REGION Network 2: CURRENT MODEL NAME SHOWN IN HMI
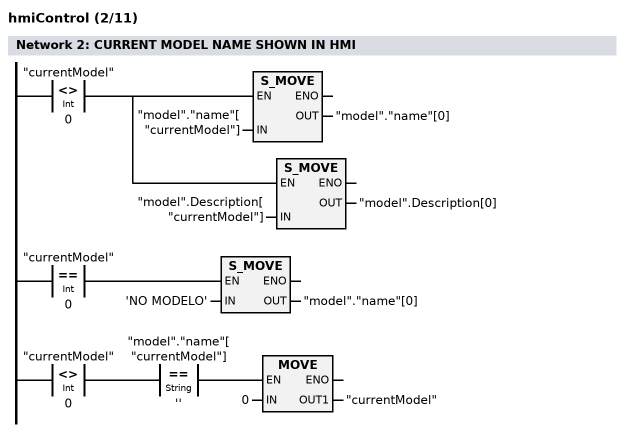
   RUNG wire#powerrail
      { S7_Templates := "SrcType := Int" } NE_Contact(in1 := "currentModel", in2 := 0)
      wire#w1
      S_Move(in := "model"."name"["currentModel"], out => "model"."name"[0])
   END_RUNG
   RUNG wire#w1
      S_Move(in := "model".Description["currentModel"], out => "model".Description[0])
   END_RUNG
   RUNG wire#powerrail
      { S7_Templates := "SrcType := Int" } EQ_Contact(in1 := "currentModel", in2 := 0)
      S_Move(in := 'NO MODELO', out => "model"."name"[0])
   END_RUNG
   RUNG wire#powerrail
      { S7_Templates := "SrcType := Int" } NE_Contact(in1 := "currentModel", in2 := 0)
      { S7_Templates := "SrcType := String" } EQ_Contact(in1 := "model"."name"["currentModel"], in2 := '')
      Move(in := 0, out1 => "currentModel")
   END_RUNG
   // the same network as SCL:
   IF "currentModel" <> 0 THEN
       "model"."name"[0] := "model"."name"["currentModel"];
       "model".Description[0] := "model".Description["currentModel"];
   END_IF;
   IF "currentModel" = 0 THEN "model"."name"[0] := 'NO MODELO'; END_IF;
   IF ("currentModel" <> 0) AND ("model"."name"["currentModel"] = '') THEN "currentModel" := 0; END_IF;
END_REGION

REGION Network 3: MODEL CHANGE (VARIABLE ACTUALIZATION)
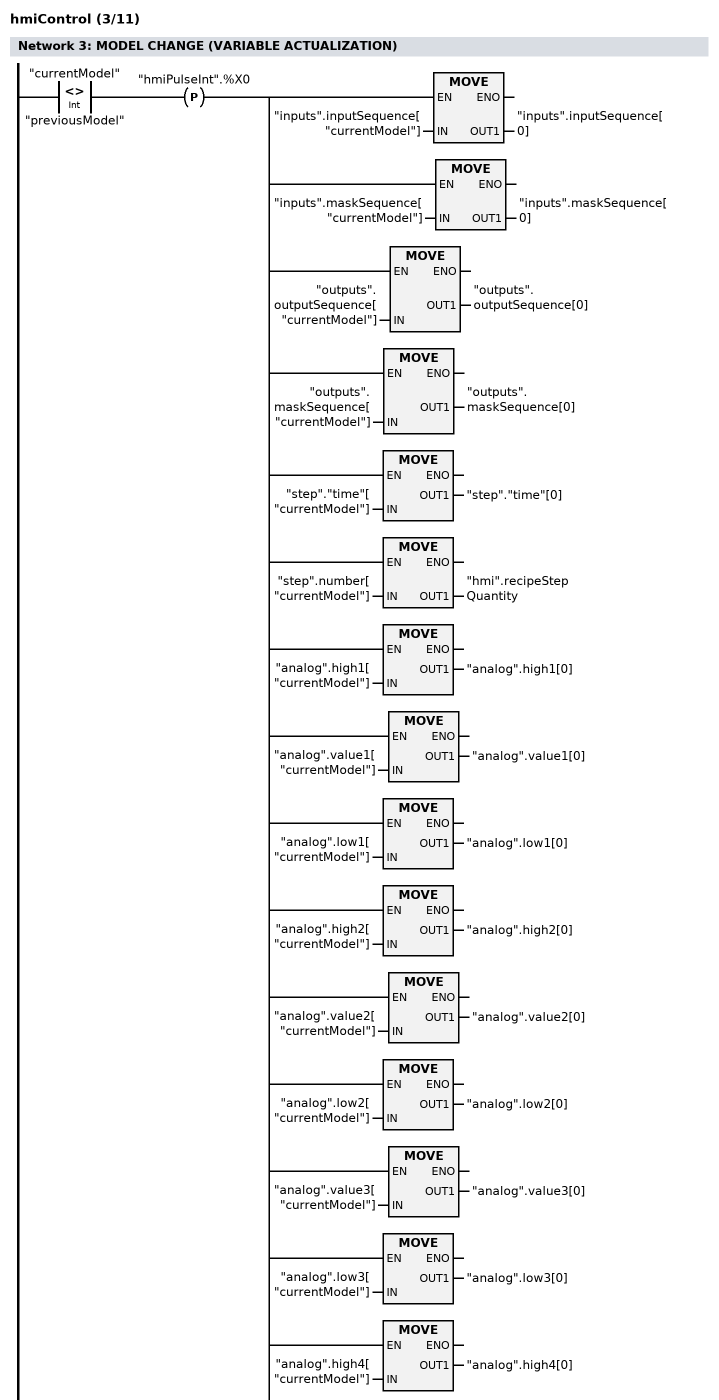
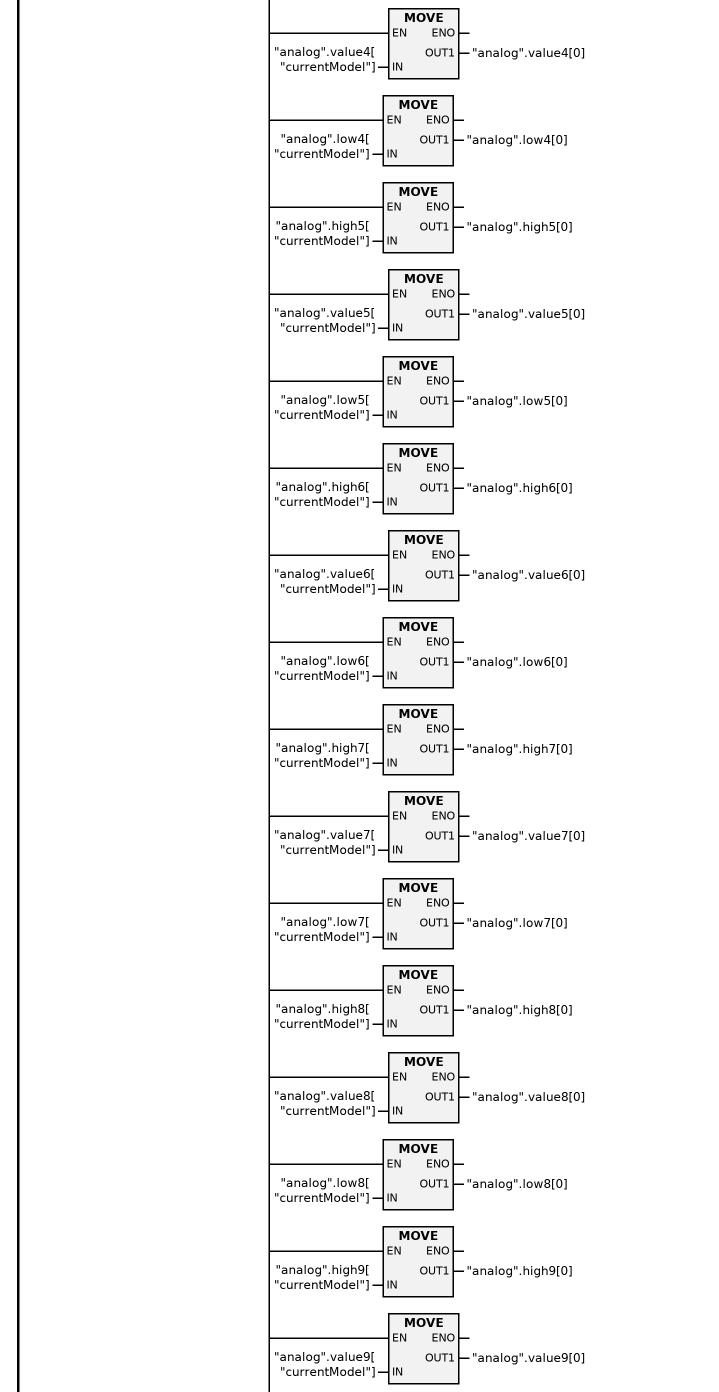
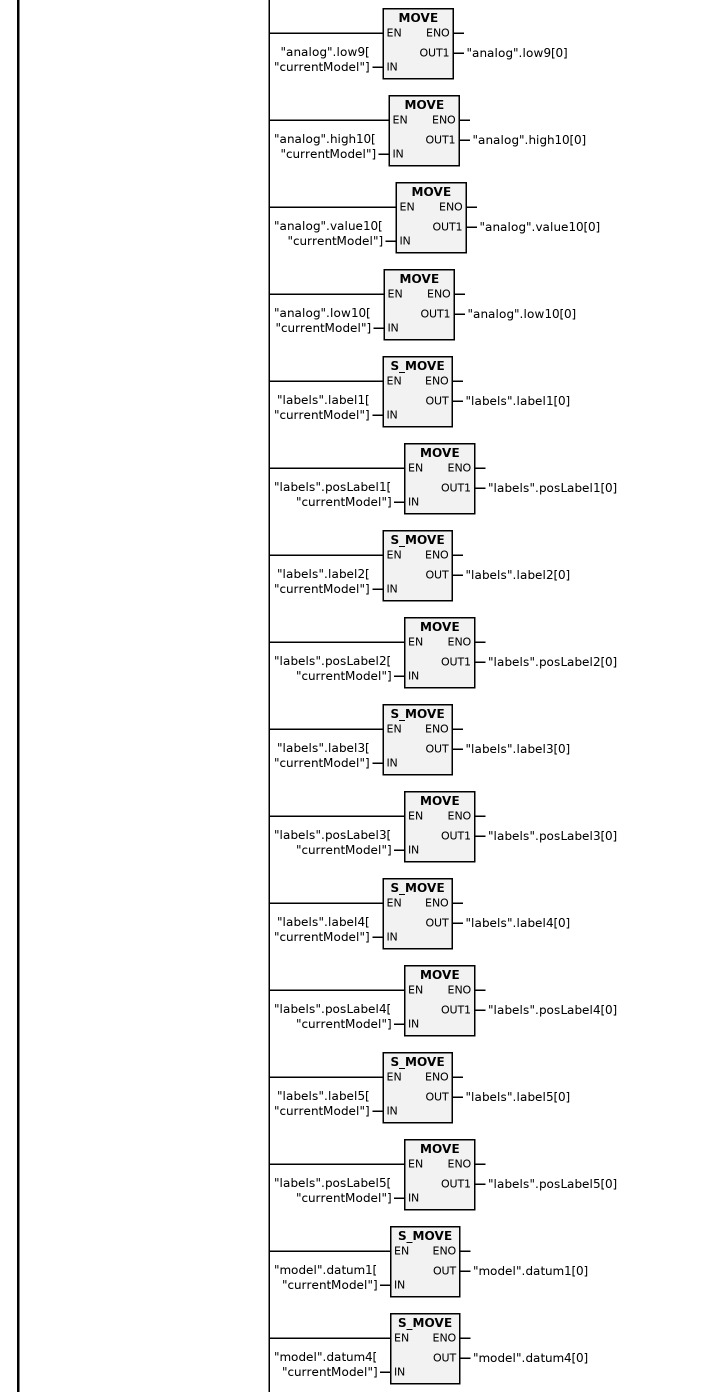
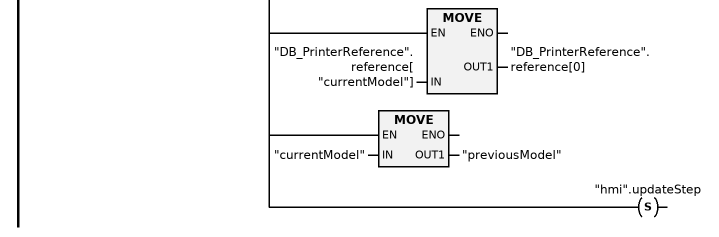
   RUNG wire#powerrail
      { S7_Templates := "SrcType := Int" } NE_Contact(in1 := "currentModel", in2 := "previousModel")
      P_Trig( "hmiPulseInt".%X0 )
      wire#w1
      Move(in := "inputs".inputSequence["currentModel"], out1 => "inputs".inputSequence[0])
   END_RUNG
   RUNG wire#w1
      Move(in := "inputs".maskSequence["currentModel"], out1 => "inputs".maskSequence[0])
   END_RUNG
   RUNG wire#w1
      Move(in := "outputs".outputSequence["currentModel"], out1 => "outputs".outputSequence[0])
   END_RUNG
   RUNG wire#w1
      Move(in := "outputs".maskSequence["currentModel"], out1 => "outputs".maskSequence[0])
   END_RUNG
   RUNG wire#w1
      Move(in := "step"."time"["currentModel"], out1 => "step"."time"[0])
   END_RUNG
   RUNG wire#w1
      Move(in := "step".number["currentModel"], out1 => "hmi".recipeStepQuantity)
   END_RUNG
   RUNG wire#w1
      Move(in := "analog".high1["currentModel"], out1 => "analog".high1[0])
   END_RUNG
   RUNG wire#w1
      Move(in := "analog".value1["currentModel"], out1 => "analog".value1[0])
   END_RUNG
   RUNG wire#w1
      Move(in := "analog".low1["currentModel"], out1 => "analog".low1[0])
   END_RUNG
   RUNG wire#w1
      Move(in := "analog".high2["currentModel"], out1 => "analog".high2[0])
   END_RUNG
   RUNG wire#w1
      Move(in := "analog".value2["currentModel"], out1 => "analog".value2[0])
   END_RUNG
   RUNG wire#w1
      Move(in := "analog".low2["currentModel"], out1 => "analog".low2[0])
   END_RUNG
   RUNG wire#w1
      Move(in := "analog".value3["currentModel"], out1 => "analog".value3[0])
   END_RUNG
   RUNG wire#w1
      Move(in := "analog".low3["currentModel"], out1 => "analog".low3[0])
   END_RUNG
   RUNG wire#w1
      Move(in := "analog".high4["currentModel"], out1 => "analog".high4[0])
   END_RUNG
   RUNG wire#w1
      Move(in := "analog".value4["currentModel"], out1 => "analog".value4[0])
   END_RUNG
   RUNG wire#w1
      Move(in := "analog".low4["currentModel"], out1 => "analog".low4[0])
   END_RUNG
   RUNG wire#w1
      Move(in := "analog".high5["currentModel"], out1 => "analog".high5[0])
   END_RUNG
   RUNG wire#w1
      Move(in := "analog".value5["currentModel"], out1 => "analog".value5[0])
   END_RUNG
   RUNG wire#w1
      Move(in := "analog".low5["currentModel"], out1 => "analog".low5[0])
   END_RUNG
   RUNG wire#w1
      Move(in := "analog".high6["currentModel"], out1 => "analog".high6[0])
   END_RUNG
   RUNG wire#w1
      Move(in := "analog".value6["currentModel"], out1 => "analog".value6[0])
   END_RUNG
   RUNG wire#w1
      Move(in := "analog".low6["currentModel"], out1 => "analog".low6[0])
   END_RUNG
   RUNG wire#w1
      Move(in := "analog".high7["currentModel"], out1 => "analog".high7[0])
   END_RUNG
   RUNG wire#w1
      Move(in := "analog".value7["currentModel"], out1 => "analog".value7[0])
   END_RUNG
   RUNG wire#w1
      Move(in := "analog".low7["currentModel"], out1 => "analog".low7[0])
   END_RUNG
   RUNG wire#w1
      Move(in := "analog".high8["currentModel"], out1 => "analog".high8[0])
   END_RUNG
   RUNG wire#w1
      Move(in := "analog".value8["currentModel"], out1 => "analog".value8[0])
   END_RUNG
   RUNG wire#w1
      Move(in := "analog".low8["currentModel"], out1 => "analog".low8[0])
   END_RUNG
   RUNG wire#w1
      Move(in := "analog".high9["currentModel"], out1 => "analog".high9[0])
   END_RUNG
   RUNG wire#w1
      Move(in := "analog".value9["currentModel"], out1 => "analog".value9[0])
   END_RUNG
   RUNG wire#w1
      Move(in := "analog".low9["currentModel"], out1 => "analog".low9[0])
   END_RUNG
   RUNG wire#w1
      Move(in := "analog".high10["currentModel"], out1 => "analog".high10[0])
   END_RUNG
   RUNG wire#w1
      Move(in := "analog".value10["currentModel"], out1 => "analog".value10[0])
   END_RUNG
   RUNG wire#w1
      Move(in := "analog".low10["currentModel"], out1 => "analog".low10[0])
   END_RUNG
   RUNG wire#w1
      S_Move(in := "labels".label1["currentModel"], out => "labels".label1[0])
   END_RUNG
   RUNG wire#w1
      Move(in := "labels".posLabel1["currentModel"], out1 => "labels".posLabel1[0])
   END_RUNG
   RUNG wire#w1
      S_Move(in := "labels".label2["currentModel"], out => "labels".label2[0])
   END_RUNG
   RUNG wire#w1
      Move(in := "labels".posLabel2["currentModel"], out1 => "labels".posLabel2[0])
   END_RUNG
   RUNG wire#w1
      S_Move(in := "labels".label3["currentModel"], out => "labels".label3[0])
   END_RUNG
   RUNG wire#w1
      Move(in := "labels".posLabel3["currentModel"], out1 => "labels".posLabel3[0])
   END_RUNG
   RUNG wire#w1
      S_Move(in := "labels".label4["currentModel"], out => "labels".label4[0])
   END_RUNG
   RUNG wire#w1
      Move(in := "labels".posLabel4["currentModel"], out1 => "labels".posLabel4[0])
   END_RUNG
   RUNG wire#w1
      S_Move(in := "labels".label5["currentModel"], out => "labels".label5[0])
   END_RUNG
   RUNG wire#w1
      Move(in := "labels".posLabel5["currentModel"], out1 => "labels".posLabel5[0])
   END_RUNG
   RUNG wire#w1
      S_Move(in := "model".datum1["currentModel"], out => "model".datum1[0])
   END_RUNG
   RUNG wire#w1
      S_Move(in := "model".datum4["currentModel"], out => "model".datum4[0])
   END_RUNG
   RUNG wire#w1
      Move(in := "DB_PrinterReference".reference["currentModel"], out1 => "DB_PrinterReference".reference[0])
   END_RUNG
   RUNG wire#w1
      Move(in := "currentModel", out1 => "previousModel")
   END_RUNG
   RUNG wire#w1
      S_Coil( "hmi".updateStep )
   END_RUNG
   // the same network as SCL:
   #_w1 := "currentModel" <> "previousModel";
   #_w2 := #_w1 AND NOT "hmiPulseInt".%X0;   // rising edge
   "hmiPulseInt".%X0 := #_w1;
   IF #_w2 THEN
       "inputs".inputSequence[0] := "inputs".inputSequence["currentModel"];
       "inputs".maskSequence[0] := "inputs".maskSequence["currentModel"];
       "outputs".outputSequence[0] := "outputs".outputSequence["currentModel"];
       "outputs".maskSequence[0] := "outputs".maskSequence["currentModel"];
       "step"."time"[0] := "step"."time"["currentModel"];
       "hmi".recipeStepQuantity := "step".number["currentModel"];
       "analog".high1[0] := "analog".high1["currentModel"];
       "analog".value1[0] := "analog".value1["currentModel"];
       "analog".low1[0] := "analog".low1["currentModel"];
       "analog".high2[0] := "analog".high2["currentModel"];
       "analog".value2[0] := "analog".value2["currentModel"];
       "analog".low2[0] := "analog".low2["currentModel"];
       "analog".value3[0] := "analog".value3["currentModel"];
       "analog".low3[0] := "analog".low3["currentModel"];
       "analog".high4[0] := "analog".high4["currentModel"];
       "analog".value4[0] := "analog".value4["currentModel"];
       "analog".low4[0] := "analog".low4["currentModel"];
       "analog".high5[0] := "analog".high5["currentModel"];
       "analog".value5[0] := "analog".value5["currentModel"];
       "analog".low5[0] := "analog".low5["currentModel"];
       "analog".high6[0] := "analog".high6["currentModel"];
       "analog".value6[0] := "analog".value6["currentModel"];
       "analog".low6[0] := "analog".low6["currentModel"];
       "analog".high7[0] := "analog".high7["currentModel"];
       "analog".value7[0] := "analog".value7["currentModel"];
       "analog".low7[0] := "analog".low7["currentModel"];
       "analog".high8[0] := "analog".high8["currentModel"];
       "analog".value8[0] := "analog".value8["currentModel"];
       "analog".low8[0] := "analog".low8["currentModel"];
       "analog".high9[0] := "analog".high9["currentModel"];
       "analog".value9[0] := "analog".value9["currentModel"];
       "analog".low9[0] := "analog".low9["currentModel"];
       "analog".high10[0] := "analog".high10["currentModel"];
       "analog".value10[0] := "analog".value10["currentModel"];
       "analog".low10[0] := "analog".low10["currentModel"];
       "labels".label1[0] := "labels".label1["currentModel"];
       "labels".posLabel1[0] := "labels".posLabel1["currentModel"];
       "labels".label2[0] := "labels".label2["currentModel"];
       "labels".posLabel2[0] := "labels".posLabel2["currentModel"];
       "labels".label3[0] := "labels".label3["currentModel"];
       "labels".posLabel3[0] := "labels".posLabel3["currentModel"];
       "labels".label4[0] := "labels".label4["currentModel"];
       "labels".posLabel4[0] := "labels".posLabel4["currentModel"];
       "labels".label5[0] := "labels".label5["currentModel"];
       "labels".posLabel5[0] := "labels".posLabel5["currentModel"];
       "model".datum1[0] := "model".datum1["currentModel"];
       "model".datum4[0] := "model".datum4["currentModel"];
       "DB_PrinterReference".reference[0] := "DB_PrinterReference".reference["currentModel"];
       "previousModel" := "currentModel";
       "hmi".updateStep := TRUE;
   END_IF;
END_REGION

REGION Network 4: STEP CHANGE IN RECIPE
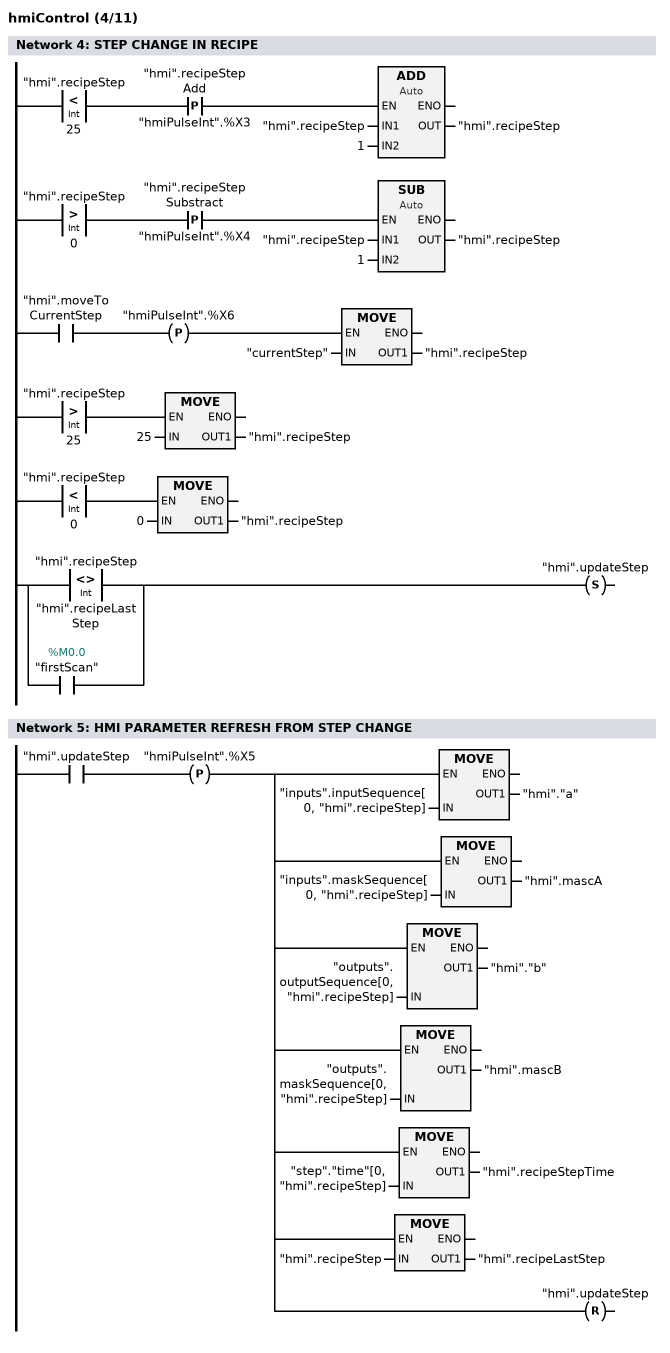
   RUNG wire#powerrail
      { S7_Templates := "SrcType := Int" } LT_Contact(in1 := "hmi".recipeStep, in2 := 25)
      P_Contact(operand := "hmi".recipeStepAdd, bit := "hmiPulseInt".%X3)
      Add(in1 := "hmi".recipeStep, in2 := 1, out => "hmi".recipeStep)
   END_RUNG
   RUNG wire#powerrail
      { S7_Templates := "SrcType := Int" } GT_Contact(in1 := "hmi".recipeStep, in2 := 0)
      P_Contact(operand := "hmi".recipeStepSubstract, bit := "hmiPulseInt".%X4)
      Sub(in1 := "hmi".recipeStep, in2 := 1, out => "hmi".recipeStep)
   END_RUNG
   RUNG wire#powerrail
      Contact( "hmi".moveToCurrentStep )
      P_Trig( "hmiPulseInt".%X6 )
      Move(in := "currentStep", out1 => "hmi".recipeStep)
   END_RUNG
   RUNG wire#powerrail
      { S7_Templates := "SrcType := Int" } GT_Contact(in1 := "hmi".recipeStep, in2 := 25)
      Move(in := 25, out1 => "hmi".recipeStep)
   END_RUNG
   RUNG wire#powerrail
      { S7_Templates := "SrcType := Int" } LT_Contact(in1 := "hmi".recipeStep, in2 := 0)
      Move(in := 0, out1 => "hmi".recipeStep)
   END_RUNG
   RUNG wire#powerrail
      { S7_Templates := "SrcType := Int" } NE_Contact(in1 := "hmi".recipeStep, in2 := "hmi".recipeLastStep)
      wire#w1
      S_Coil( "hmi".updateStep )
   END_RUNG
   RUNG wire#powerrail
      Contact( "firstScan" )
   END_RUNG wire#w1
   // the same network as SCL:
   #_w1 := ("hmi".recipeStep < 25) AND "hmi".recipeStepAdd AND NOT "hmiPulseInt".%X3;   // rising edge of "hmi".recipeStepAdd
   "hmiPulseInt".%X3 := "hmi".recipeStepAdd;
   IF #_w1 THEN "hmi".recipeStep := "hmi".recipeStep + 1; END_IF;
   #_w2 := ("hmi".recipeStep > 0) AND "hmi".recipeStepSubstract AND NOT "hmiPulseInt".%X4;   // rising edge of "hmi".recipeStepSubstract
   "hmiPulseInt".%X4 := "hmi".recipeStepSubstract;
   IF #_w2 THEN "hmi".recipeStep := "hmi".recipeStep - 1; END_IF;
   #_w3 := "hmi".moveToCurrentStep AND NOT "hmiPulseInt".%X6;   // rising edge
   "hmiPulseInt".%X6 := "hmi".moveToCurrentStep;
   IF #_w3 THEN "hmi".recipeStep := "currentStep"; END_IF;
   IF "hmi".recipeStep > 25 THEN "hmi".recipeStep := 25; END_IF;
   IF "hmi".recipeStep < 0 THEN "hmi".recipeStep := 0; END_IF;
   IF ("hmi".recipeStep <> "hmi".recipeLastStep) OR "firstScan" THEN "hmi".updateStep := TRUE; END_IF;
END_REGION

REGION Network 5: HMI PARAMETER REFRESH FROM STEP CHANGE
   RUNG wire#powerrail
      Contact( "hmi".updateStep )
      P_Trig( "hmiPulseInt".%X5 )
      wire#w1
      Move(in := "inputs".inputSequence[0, "hmi".recipeStep], out1 => "hmi"."a")
   END_RUNG
   RUNG wire#w1
      Move(in := "inputs".maskSequence[0, "hmi".recipeStep], out1 => "hmi".mascA)
   END_RUNG
   RUNG wire#w1
      Move(in := "outputs".outputSequence[0, "hmi".recipeStep], out1 => "hmi"."b")
   END_RUNG
   RUNG wire#w1
      Move(in := "outputs".maskSequence[0, "hmi".recipeStep], out1 => "hmi".mascB)
   END_RUNG
   RUNG wire#w1
      Move(in := "step"."time"[0, "hmi".recipeStep], out1 => "hmi".recipeStepTime)
   END_RUNG
   RUNG wire#w1
      Move(in := "hmi".recipeStep, out1 => "hmi".recipeLastStep)
   END_RUNG
   RUNG wire#w1
      R_Coil( "hmi".updateStep )
   END_RUNG
   // the same network as SCL:
   #_w1 := "hmi".updateStep AND NOT "hmiPulseInt".%X5;   // rising edge
   "hmiPulseInt".%X5 := "hmi".updateStep;
   IF #_w1 THEN
       "hmi"."a" := "inputs".inputSequence[0, "hmi".recipeStep];
       "hmi".mascA := "inputs".maskSequence[0, "hmi".recipeStep];
       "hmi"."b" := "outputs".outputSequence[0, "hmi".recipeStep];
       "hmi".mascB := "outputs".maskSequence[0, "hmi".recipeStep];
       "hmi".recipeStepTime := "step"."time"[0, "hmi".recipeStep];
       "hmi".recipeLastStep := "hmi".recipeStep;
       "hmi".updateStep := FALSE;
   END_IF;
END_REGION

REGION Network 6: EDIT VALUES IN CURRENT RECIPE
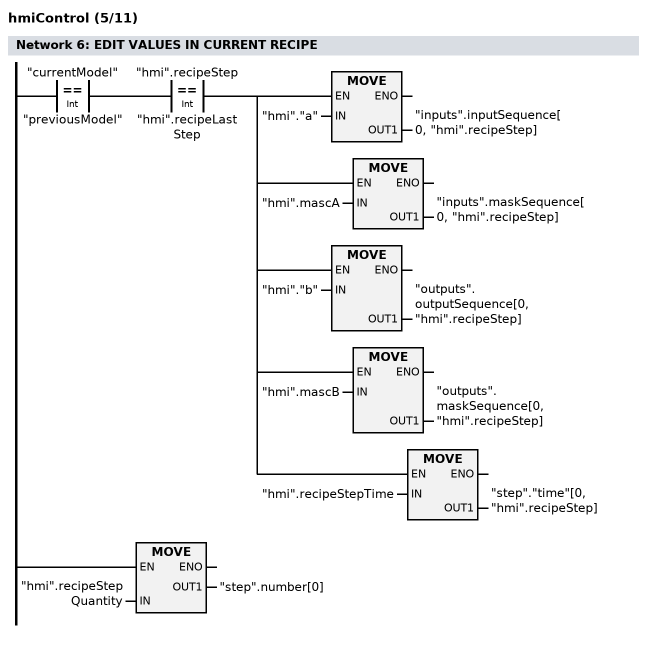
   RUNG wire#powerrail
      { S7_Templates := "SrcType := Int" } EQ_Contact(in1 := "currentModel", in2 := "previousModel")
      { S7_Templates := "SrcType := Int" } EQ_Contact(in1 := "hmi".recipeStep, in2 := "hmi".recipeLastStep)
      wire#w1
      Move(in := "hmi"."a", out1 => "inputs".inputSequence[0, "hmi".recipeStep])
   END_RUNG
   RUNG wire#w1
      Move(in := "hmi".mascA, out1 => "inputs".maskSequence[0, "hmi".recipeStep])
   END_RUNG
   RUNG wire#w1
      Move(in := "hmi"."b", out1 => "outputs".outputSequence[0, "hmi".recipeStep])
   END_RUNG
   RUNG wire#w1
      Move(in := "hmi".mascB, out1 => "outputs".maskSequence[0, "hmi".recipeStep])
   END_RUNG
   RUNG wire#w1
      Move(in := "hmi".recipeStepTime, out1 => "step"."time"[0, "hmi".recipeStep])
   END_RUNG
   RUNG wire#powerrail
      Move(in := "hmi".recipeStepQuantity, out1 => "step".number[0])
   END_RUNG
   // the same network as SCL:
   #_w1 := ("currentModel" = "previousModel") AND ("hmi".recipeStep = "hmi".recipeLastStep);
   IF #_w1 THEN
       "inputs".inputSequence[0, "hmi".recipeStep] := "hmi"."a";
       "inputs".maskSequence[0, "hmi".recipeStep] := "hmi".mascA;
       "outputs".outputSequence[0, "hmi".recipeStep] := "hmi"."b";
       "outputs".maskSequence[0, "hmi".recipeStep] := "hmi".mascB;
       "step"."time"[0, "hmi".recipeStep] := "hmi".recipeStepTime;
   END_IF;
   "step".number[0] := "hmi".recipeStepQuantity;
END_REGION

REGION Network 7: WRITE AND READ IN SCREEN
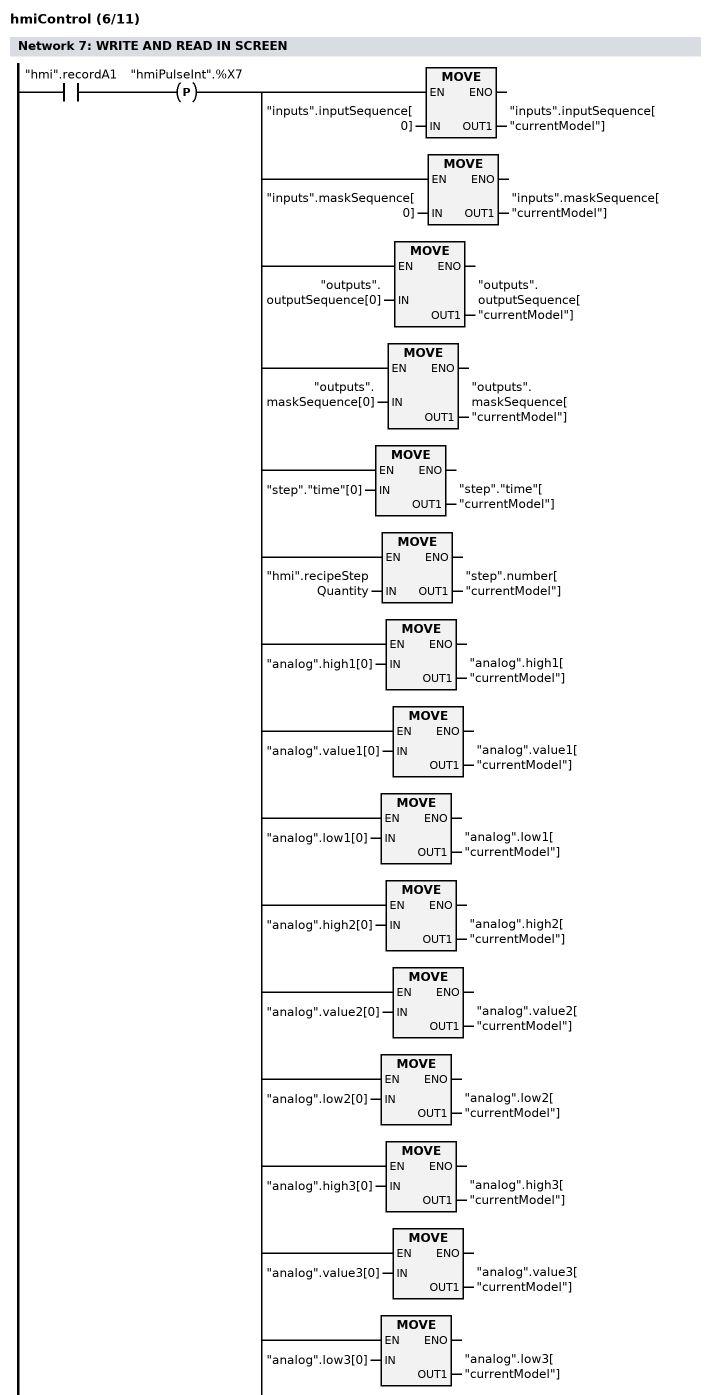
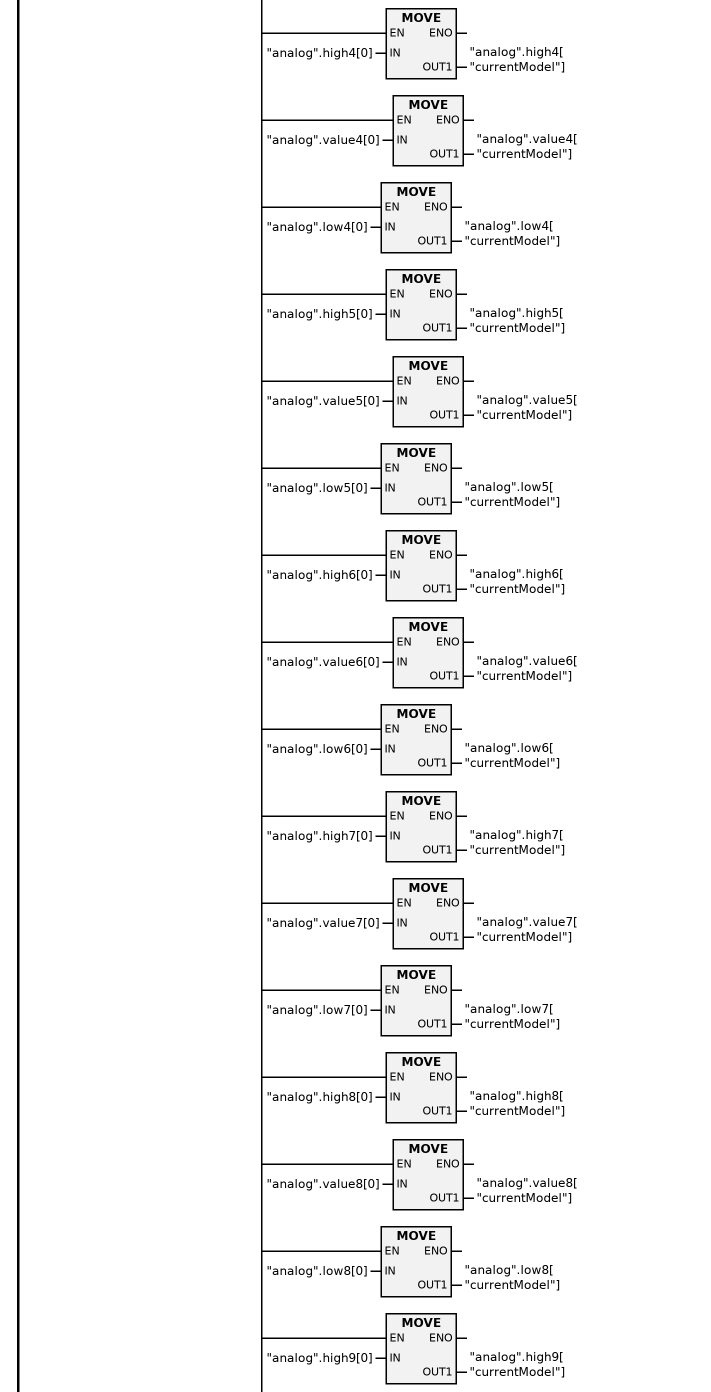
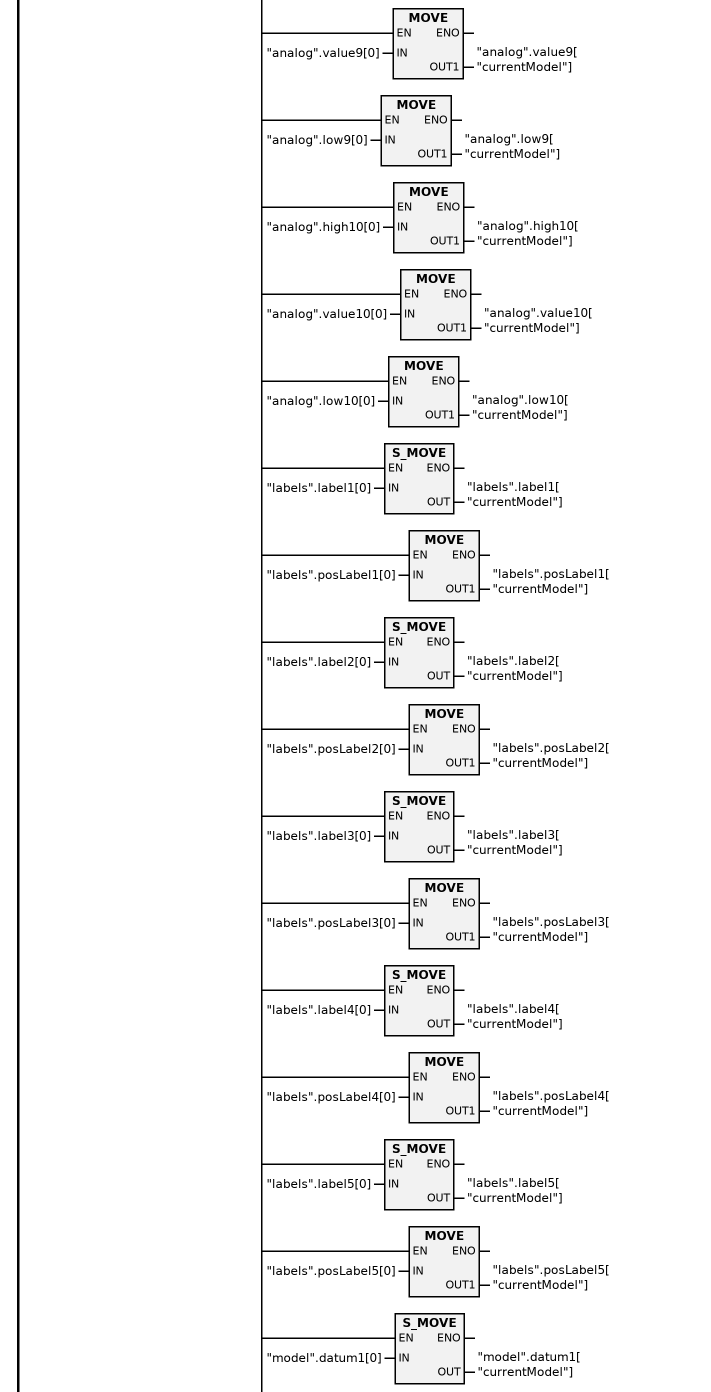
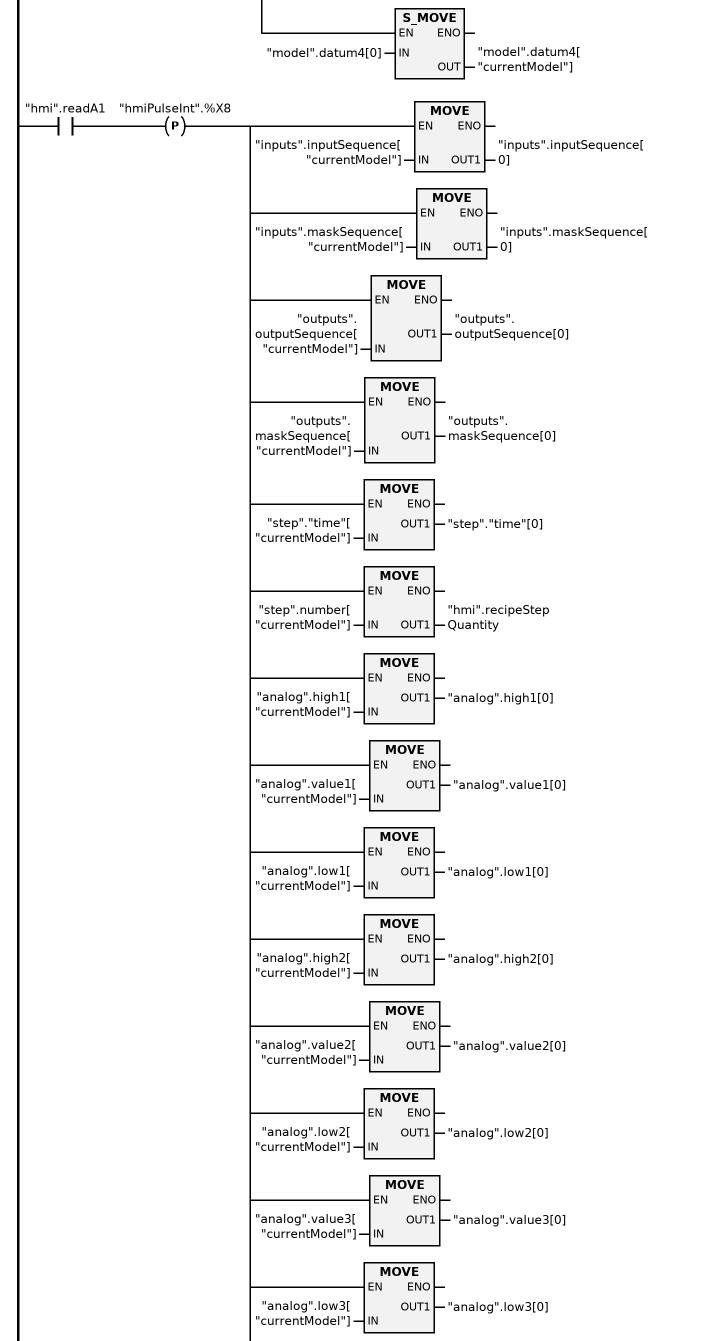
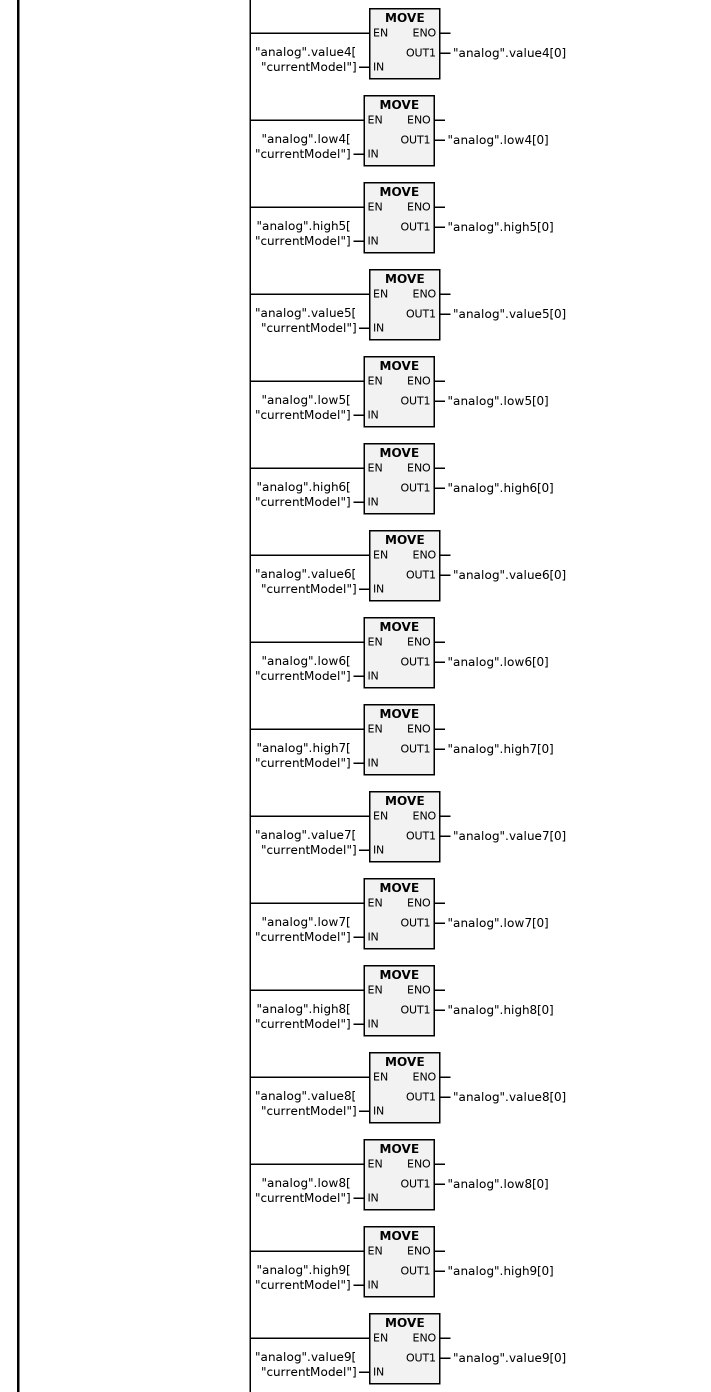
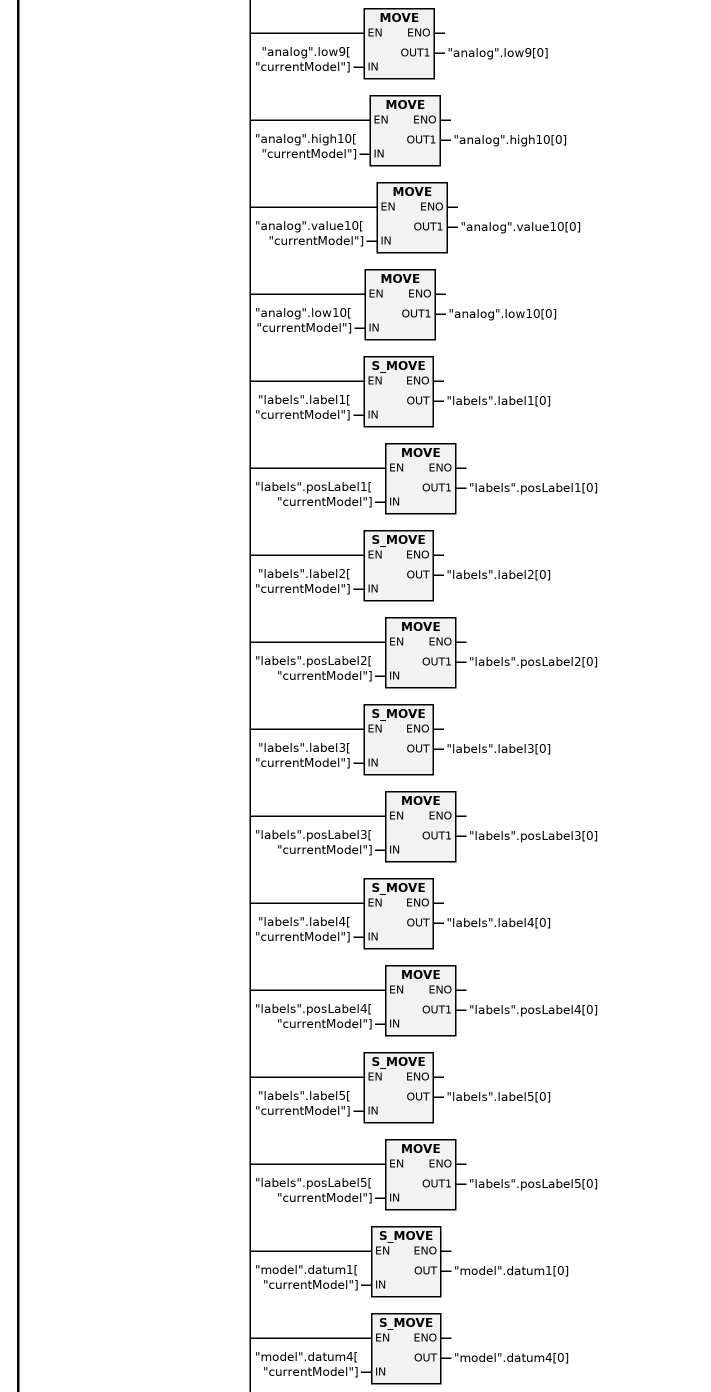
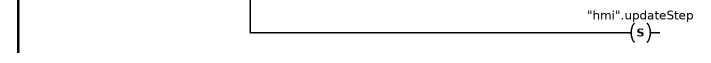
   RUNG wire#powerrail
      Contact( "hmi".recordA1 )
      P_Trig( "hmiPulseInt".%X7 )
      wire#w1
      Move(in := "inputs".inputSequence[0], out1 => "inputs".inputSequence["currentModel"])
   END_RUNG
   RUNG wire#w1
      Move(in := "inputs".maskSequence[0], out1 => "inputs".maskSequence["currentModel"])
   END_RUNG
   RUNG wire#w1
      Move(in := "outputs".outputSequence[0], out1 => "outputs".outputSequence["currentModel"])
   END_RUNG
   RUNG wire#w1
      Move(in := "outputs".maskSequence[0], out1 => "outputs".maskSequence["currentModel"])
   END_RUNG
   RUNG wire#w1
      Move(in := "step"."time"[0], out1 => "step"."time"["currentModel"])
   END_RUNG
   RUNG wire#w1
      Move(in := "hmi".recipeStepQuantity, out1 => "step".number["currentModel"])
   END_RUNG
   RUNG wire#w1
      Move(in := "analog".high1[0], out1 => "analog".high1["currentModel"])
   END_RUNG
   RUNG wire#w1
      Move(in := "analog".value1[0], out1 => "analog".value1["currentModel"])
   END_RUNG
   RUNG wire#w1
      Move(in := "analog".low1[0], out1 => "analog".low1["currentModel"])
   END_RUNG
   RUNG wire#w1
      Move(in := "analog".high2[0], out1 => "analog".high2["currentModel"])
   END_RUNG
   RUNG wire#w1
      Move(in := "analog".value2[0], out1 => "analog".value2["currentModel"])
   END_RUNG
   RUNG wire#w1
      Move(in := "analog".low2[0], out1 => "analog".low2["currentModel"])
   END_RUNG
   RUNG wire#w1
      Move(in := "analog".high3[0], out1 => "analog".high3["currentModel"])
   END_RUNG
   RUNG wire#w1
      Move(in := "analog".value3[0], out1 => "analog".value3["currentModel"])
   END_RUNG
   RUNG wire#w1
      Move(in := "analog".low3[0], out1 => "analog".low3["currentModel"])
   END_RUNG
   RUNG wire#w1
      Move(in := "analog".high4[0], out1 => "analog".high4["currentModel"])
   END_RUNG
   RUNG wire#w1
      Move(in := "analog".value4[0], out1 => "analog".value4["currentModel"])
   END_RUNG
   RUNG wire#w1
      Move(in := "analog".low4[0], out1 => "analog".low4["currentModel"])
   END_RUNG
   RUNG wire#w1
      Move(in := "analog".high5[0], out1 => "analog".high5["currentModel"])
   END_RUNG
   RUNG wire#w1
      Move(in := "analog".value5[0], out1 => "analog".value5["currentModel"])
   END_RUNG
   RUNG wire#w1
      Move(in := "analog".low5[0], out1 => "analog".low5["currentModel"])
   END_RUNG
   RUNG wire#w1
      Move(in := "analog".high6[0], out1 => "analog".high6["currentModel"])
   END_RUNG
   RUNG wire#w1
      Move(in := "analog".value6[0], out1 => "analog".value6["currentModel"])
   END_RUNG
   RUNG wire#w1
      Move(in := "analog".low6[0], out1 => "analog".low6["currentModel"])
   END_RUNG
   RUNG wire#w1
      Move(in := "analog".high7[0], out1 => "analog".high7["currentModel"])
   END_RUNG
   RUNG wire#w1
      Move(in := "analog".value7[0], out1 => "analog".value7["currentModel"])
   END_RUNG
   RUNG wire#w1
      Move(in := "analog".low7[0], out1 => "analog".low7["currentModel"])
   END_RUNG
   RUNG wire#w1
      Move(in := "analog".high8[0], out1 => "analog".high8["currentModel"])
   END_RUNG
   RUNG wire#w1
      Move(in := "analog".value8[0], out1 => "analog".value8["currentModel"])
   END_RUNG
   RUNG wire#w1
      Move(in := "analog".low8[0], out1 => "analog".low8["currentModel"])
   END_RUNG
   RUNG wire#w1
      Move(in := "analog".high9[0], out1 => "analog".high9["currentModel"])
   END_RUNG
   RUNG wire#w1
      Move(in := "analog".value9[0], out1 => "analog".value9["currentModel"])
   END_RUNG
   RUNG wire#w1
      Move(in := "analog".low9[0], out1 => "analog".low9["currentModel"])
   END_RUNG
   RUNG wire#w1
      Move(in := "analog".high10[0], out1 => "analog".high10["currentModel"])
   END_RUNG
   RUNG wire#w1
      Move(in := "analog".value10[0], out1 => "analog".value10["currentModel"])
   END_RUNG
   RUNG wire#w1
      Move(in := "analog".low10[0], out1 => "analog".low10["currentModel"])
   END_RUNG
   RUNG wire#w1
      S_Move(in := "labels".label1[0], out => "labels".label1["currentModel"])
   END_RUNG
   RUNG wire#w1
      Move(in := "labels".posLabel1[0], out1 => "labels".posLabel1["currentModel"])
   END_RUNG
   RUNG wire#w1
      S_Move(in := "labels".label2[0], out => "labels".label2["currentModel"])
   END_RUNG
   RUNG wire#w1
      Move(in := "labels".posLabel2[0], out1 => "labels".posLabel2["currentModel"])
   END_RUNG
   RUNG wire#w1
      S_Move(in := "labels".label3[0], out => "labels".label3["currentModel"])
   END_RUNG
   RUNG wire#w1
      Move(in := "labels".posLabel3[0], out1 => "labels".posLabel3["currentModel"])
   END_RUNG
   RUNG wire#w1
      S_Move(in := "labels".label4[0], out => "labels".label4["currentModel"])
   END_RUNG
   RUNG wire#w1
      Move(in := "labels".posLabel4[0], out1 => "labels".posLabel4["currentModel"])
   END_RUNG
   RUNG wire#w1
      S_Move(in := "labels".label5[0], out => "labels".label5["currentModel"])
   END_RUNG
   RUNG wire#w1
      Move(in := "labels".posLabel5[0], out1 => "labels".posLabel5["currentModel"])
   END_RUNG
   RUNG wire#w1
      S_Move(in := "model".datum1[0], out => "model".datum1["currentModel"])
   END_RUNG
   RUNG wire#w1
      S_Move(in := "model".datum4[0], out => "model".datum4["currentModel"])
   END_RUNG
   RUNG wire#powerrail
      Contact( "hmi".readA1 )
      P_Trig( "hmiPulseInt".%X8 )
      wire#w2
      Move(in := "inputs".inputSequence["currentModel"], out1 => "inputs".inputSequence[0])
   END_RUNG
   RUNG wire#w2
      Move(in := "inputs".maskSequence["currentModel"], out1 => "inputs".maskSequence[0])
   END_RUNG
   RUNG wire#w2
      Move(in := "outputs".outputSequence["currentModel"], out1 => "outputs".outputSequence[0])
   END_RUNG
   RUNG wire#w2
      Move(in := "outputs".maskSequence["currentModel"], out1 => "outputs".maskSequence[0])
   END_RUNG
   RUNG wire#w2
      Move(in := "step"."time"["currentModel"], out1 => "step"."time"[0])
   END_RUNG
   RUNG wire#w2
      Move(in := "step".number["currentModel"], out1 => "hmi".recipeStepQuantity)
   END_RUNG
   RUNG wire#w2
      Move(in := "analog".high1["currentModel"], out1 => "analog".high1[0])
   END_RUNG
   RUNG wire#w2
      Move(in := "analog".value1["currentModel"], out1 => "analog".value1[0])
   END_RUNG
   RUNG wire#w2
      Move(in := "analog".low1["currentModel"], out1 => "analog".low1[0])
   END_RUNG
   RUNG wire#w2
      Move(in := "analog".high2["currentModel"], out1 => "analog".high2[0])
   END_RUNG
   RUNG wire#w2
      Move(in := "analog".value2["currentModel"], out1 => "analog".value2[0])
   END_RUNG
   RUNG wire#w2
      Move(in := "analog".low2["currentModel"], out1 => "analog".low2[0])
   END_RUNG
   RUNG wire#w2
      Move(in := "analog".value3["currentModel"], out1 => "analog".value3[0])
   END_RUNG
   RUNG wire#w2
      Move(in := "analog".low3["currentModel"], out1 => "analog".low3[0])
   END_RUNG
   RUNG wire#w2
      Move(in := "analog".value4["currentModel"], out1 => "analog".value4[0])
   END_RUNG
   RUNG wire#w2
      Move(in := "analog".low4["currentModel"], out1 => "analog".low4[0])
   END_RUNG
   RUNG wire#w2
      Move(in := "analog".high5["currentModel"], out1 => "analog".high5[0])
   END_RUNG
   RUNG wire#w2
      Move(in := "analog".value5["currentModel"], out1 => "analog".value5[0])
   END_RUNG
   RUNG wire#w2
      Move(in := "analog".low5["currentModel"], out1 => "analog".low5[0])
   END_RUNG
   RUNG wire#w2
      Move(in := "analog".high6["currentModel"], out1 => "analog".high6[0])
   END_RUNG
   RUNG wire#w2
      Move(in := "analog".value6["currentModel"], out1 => "analog".value6[0])
   END_RUNG
   RUNG wire#w2
      Move(in := "analog".low6["currentModel"], out1 => "analog".low6[0])
   END_RUNG
   RUNG wire#w2
      Move(in := "analog".high7["currentModel"], out1 => "analog".high7[0])
   END_RUNG
   RUNG wire#w2
      Move(in := "analog".value7["currentModel"], out1 => "analog".value7[0])
   END_RUNG
   RUNG wire#w2
      Move(in := "analog".low7["currentModel"], out1 => "analog".low7[0])
   END_RUNG
   RUNG wire#w2
      Move(in := "analog".high8["currentModel"], out1 => "analog".high8[0])
   END_RUNG
   RUNG wire#w2
      Move(in := "analog".value8["currentModel"], out1 => "analog".value8[0])
   END_RUNG
   RUNG wire#w2
      Move(in := "analog".low8["currentModel"], out1 => "analog".low8[0])
   END_RUNG
   RUNG wire#w2
      Move(in := "analog".high9["currentModel"], out1 => "analog".high9[0])
   END_RUNG
   RUNG wire#w2
      Move(in := "analog".value9["currentModel"], out1 => "analog".value9[0])
   END_RUNG
   RUNG wire#w2
      Move(in := "analog".low9["currentModel"], out1 => "analog".low9[0])
   END_RUNG
   RUNG wire#w2
      Move(in := "analog".high10["currentModel"], out1 => "analog".high10[0])
   END_RUNG
   RUNG wire#w2
      Move(in := "analog".value10["currentModel"], out1 => "analog".value10[0])
   END_RUNG
   RUNG wire#w2
      Move(in := "analog".low10["currentModel"], out1 => "analog".low10[0])
   END_RUNG
   RUNG wire#w2
      S_Move(in := "labels".label1["currentModel"], out => "labels".label1[0])
   END_RUNG
   RUNG wire#w2
      Move(in := "labels".posLabel1["currentModel"], out1 => "labels".posLabel1[0])
   END_RUNG
   RUNG wire#w2
      S_Move(in := "labels".label2["currentModel"], out => "labels".label2[0])
   END_RUNG
   RUNG wire#w2
      Move(in := "labels".posLabel2["currentModel"], out1 => "labels".posLabel2[0])
   END_RUNG
   RUNG wire#w2
      S_Move(in := "labels".label3["currentModel"], out => "labels".label3[0])
   END_RUNG
   RUNG wire#w2
      Move(in := "labels".posLabel3["currentModel"], out1 => "labels".posLabel3[0])
   END_RUNG
   RUNG wire#w2
      S_Move(in := "labels".label4["currentModel"], out => "labels".label4[0])
   END_RUNG
   RUNG wire#w2
      Move(in := "labels".posLabel4["currentModel"], out1 => "labels".posLabel4[0])
   END_RUNG
   RUNG wire#w2
      S_Move(in := "labels".label5["currentModel"], out => "labels".label5[0])
   END_RUNG
   RUNG wire#w2
      Move(in := "labels".posLabel5["currentModel"], out1 => "labels".posLabel5[0])
   END_RUNG
   RUNG wire#w2
      S_Move(in := "model".datum1["currentModel"], out => "model".datum1[0])
   END_RUNG
   RUNG wire#w2
      S_Move(in := "model".datum4["currentModel"], out => "model".datum4[0])
   END_RUNG
   RUNG wire#w2
      S_Coil( "hmi".updateStep )
   END_RUNG
   // the same network as SCL:
   #_w1 := "hmi".recordA1 AND NOT "hmiPulseInt".%X7;   // rising edge
   "hmiPulseInt".%X7 := "hmi".recordA1;
   IF #_w1 THEN
       "inputs".inputSequence["currentModel"] := "inputs".inputSequence[0];
       "inputs".maskSequence["currentModel"] := "inputs".maskSequence[0];
       "outputs".outputSequence["currentModel"] := "outputs".outputSequence[0];
       "outputs".maskSequence["currentModel"] := "outputs".maskSequence[0];
       "step"."time"["currentModel"] := "step"."time"[0];
       "step".number["currentModel"] := "hmi".recipeStepQuantity;
       "analog".high1["currentModel"] := "analog".high1[0];
       "analog".value1["currentModel"] := "analog".value1[0];
       "analog".low1["currentModel"] := "analog".low1[0];
       "analog".high2["currentModel"] := "analog".high2[0];
       "analog".value2["currentModel"] := "analog".value2[0];
       "analog".low2["currentModel"] := "analog".low2[0];
       "analog".high3["currentModel"] := "analog".high3[0];
       "analog".value3["currentModel"] := "analog".value3[0];
       "analog".low3["currentModel"] := "analog".low3[0];
       "analog".high4["currentModel"] := "analog".high4[0];
       "analog".value4["currentModel"] := "analog".value4[0];
       "analog".low4["currentModel"] := "analog".low4[0];
       "analog".high5["currentModel"] := "analog".high5[0];
       "analog".value5["currentModel"] := "analog".value5[0];
       "analog".low5["currentModel"] := "analog".low5[0];
       "analog".high6["currentModel"] := "analog".high6[0];
       "analog".value6["currentModel"] := "analog".value6[0];
       "analog".low6["currentModel"] := "analog".low6[0];
       "analog".high7["currentModel"] := "analog".high7[0];
       "analog".value7["currentModel"] := "analog".value7[0];
       "analog".low7["currentModel"] := "analog".low7[0];
       "analog".high8["currentModel"] := "analog".high8[0];
       "analog".value8["currentModel"] := "analog".value8[0];
       "analog".low8["currentModel"] := "analog".low8[0];
       "analog".high9["currentModel"] := "analog".high9[0];
       "analog".value9["currentModel"] := "analog".value9[0];
       "analog".low9["currentModel"] := "analog".low9[0];
       "analog".high10["currentModel"] := "analog".high10[0];
       "analog".value10["currentModel"] := "analog".value10[0];
       "analog".low10["currentModel"] := "analog".low10[0];
       "labels".label1["currentModel"] := "labels".label1[0];
       "labels".posLabel1["currentModel"] := "labels".posLabel1[0];
       "labels".label2["currentModel"] := "labels".label2[0];
       "labels".posLabel2["currentModel"] := "labels".posLabel2[0];
       "labels".label3["currentModel"] := "labels".label3[0];
       "labels".posLabel3["currentModel"] := "labels".posLabel3[0];
       "labels".label4["currentModel"] := "labels".label4[0];
       "labels".posLabel4["currentModel"] := "labels".posLabel4[0];
       "labels".label5["currentModel"] := "labels".label5[0];
       "labels".posLabel5["currentModel"] := "labels".posLabel5[0];
       "model".datum1["currentModel"] := "model".datum1[0];
       "model".datum4["currentModel"] := "model".datum4[0];
   END_IF;
   #_w2 := "hmi".readA1 AND NOT "hmiPulseInt".%X8;   // rising edge
   "hmiPulseInt".%X8 := "hmi".readA1;
   IF #_w2 THEN
       "inputs".inputSequence[0] := "inputs".inputSequence["currentModel"];
       "inputs".maskSequence[0] := "inputs".maskSequence["currentModel"];
       "outputs".outputSequence[0] := "outputs".outputSequence["currentModel"];
       "outputs".maskSequence[0] := "outputs".maskSequence["currentModel"];
       "step"."time"[0] := "step"."time"["currentModel"];
       "hmi".recipeStepQuantity := "step".number["currentModel"];
       "analog".high1[0] := "analog".high1["currentModel"];
       "analog".value1[0] := "analog".value1["currentModel"];
       "analog".low1[0] := "analog".low1["currentModel"];
       "analog".high2[0] := "analog".high2["currentModel"];
       "analog".value2[0] := "analog".value2["currentModel"];
       "analog".low2[0] := "analog".low2["currentModel"];
       "analog".value3[0] := "analog".value3["currentModel"];
       "analog".low3[0] := "analog".low3["currentModel"];
       "analog".value4[0] := "analog".value4["currentModel"];
       "analog".low4[0] := "analog".low4["currentModel"];
       "analog".high5[0] := "analog".high5["currentModel"];
       "analog".value5[0] := "analog".value5["currentModel"];
       "analog".low5[0] := "analog".low5["currentModel"];
       "analog".high6[0] := "analog".high6["currentModel"];
       "analog".value6[0] := "analog".value6["currentModel"];
       "analog".low6[0] := "analog".low6["currentModel"];
       "analog".high7[0] := "analog".high7["currentModel"];
       "analog".value7[0] := "analog".value7["currentModel"];
       "analog".low7[0] := "analog".low7["currentModel"];
       "analog".high8[0] := "analog".high8["currentModel"];
       "analog".value8[0] := "analog".value8["currentModel"];
       "analog".low8[0] := "analog".low8["currentModel"];
       "analog".high9[0] := "analog".high9["currentModel"];
       "analog".value9[0] := "analog".value9["currentModel"];
       "analog".low9[0] := "analog".low9["currentModel"];
       "analog".high10[0] := "analog".high10["currentModel"];
       "analog".value10[0] := "analog".value10["currentModel"];
       "analog".low10[0] := "analog".low10["currentModel"];
       "labels".label1[0] := "labels".label1["currentModel"];
       "labels".posLabel1[0] := "labels".posLabel1["currentModel"];
       "labels".label2[0] := "labels".label2["currentModel"];
       "labels".posLabel2[0] := "labels".posLabel2["currentModel"];
       "labels".label3[0] := "labels".label3["currentModel"];
       "labels".posLabel3[0] := "labels".posLabel3["currentModel"];
       "labels".label4[0] := "labels".label4["currentModel"];
       "labels".posLabel4[0] := "labels".posLabel4["currentModel"];
       "labels".label5[0] := "labels".label5["currentModel"];
       "labels".posLabel5[0] := "labels".posLabel5["currentModel"];
       "model".datum1[0] := "model".datum1["currentModel"];
       "model".datum4[0] := "model".datum4["currentModel"];
       "hmi".updateStep := TRUE;
   END_IF;
END_REGION

REGION Network 8: NUMBER OF STEPS OF RECIPE
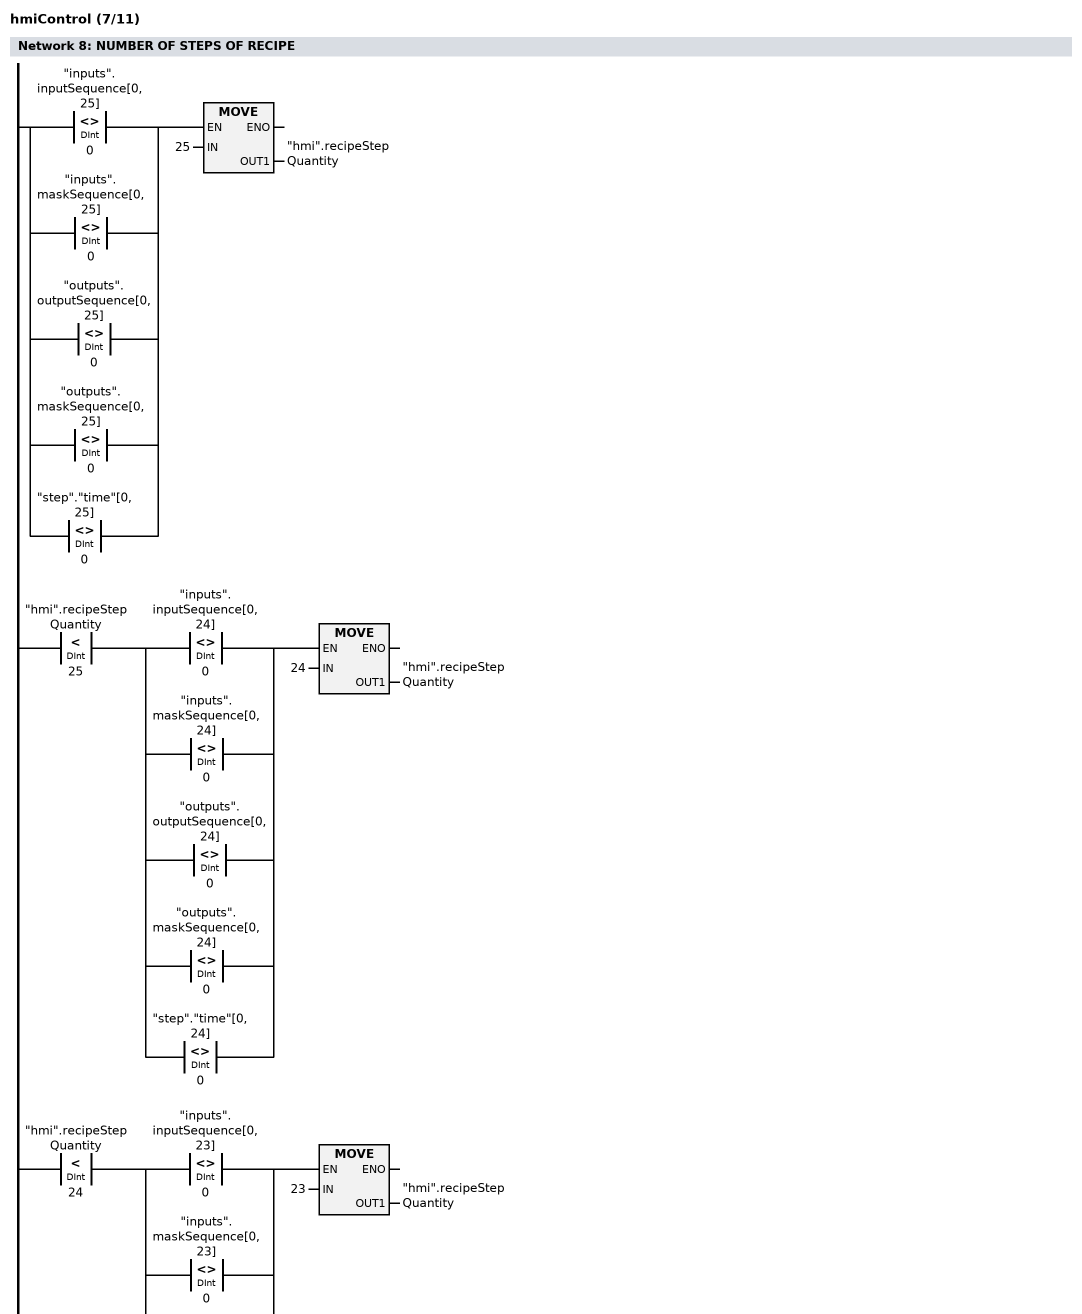
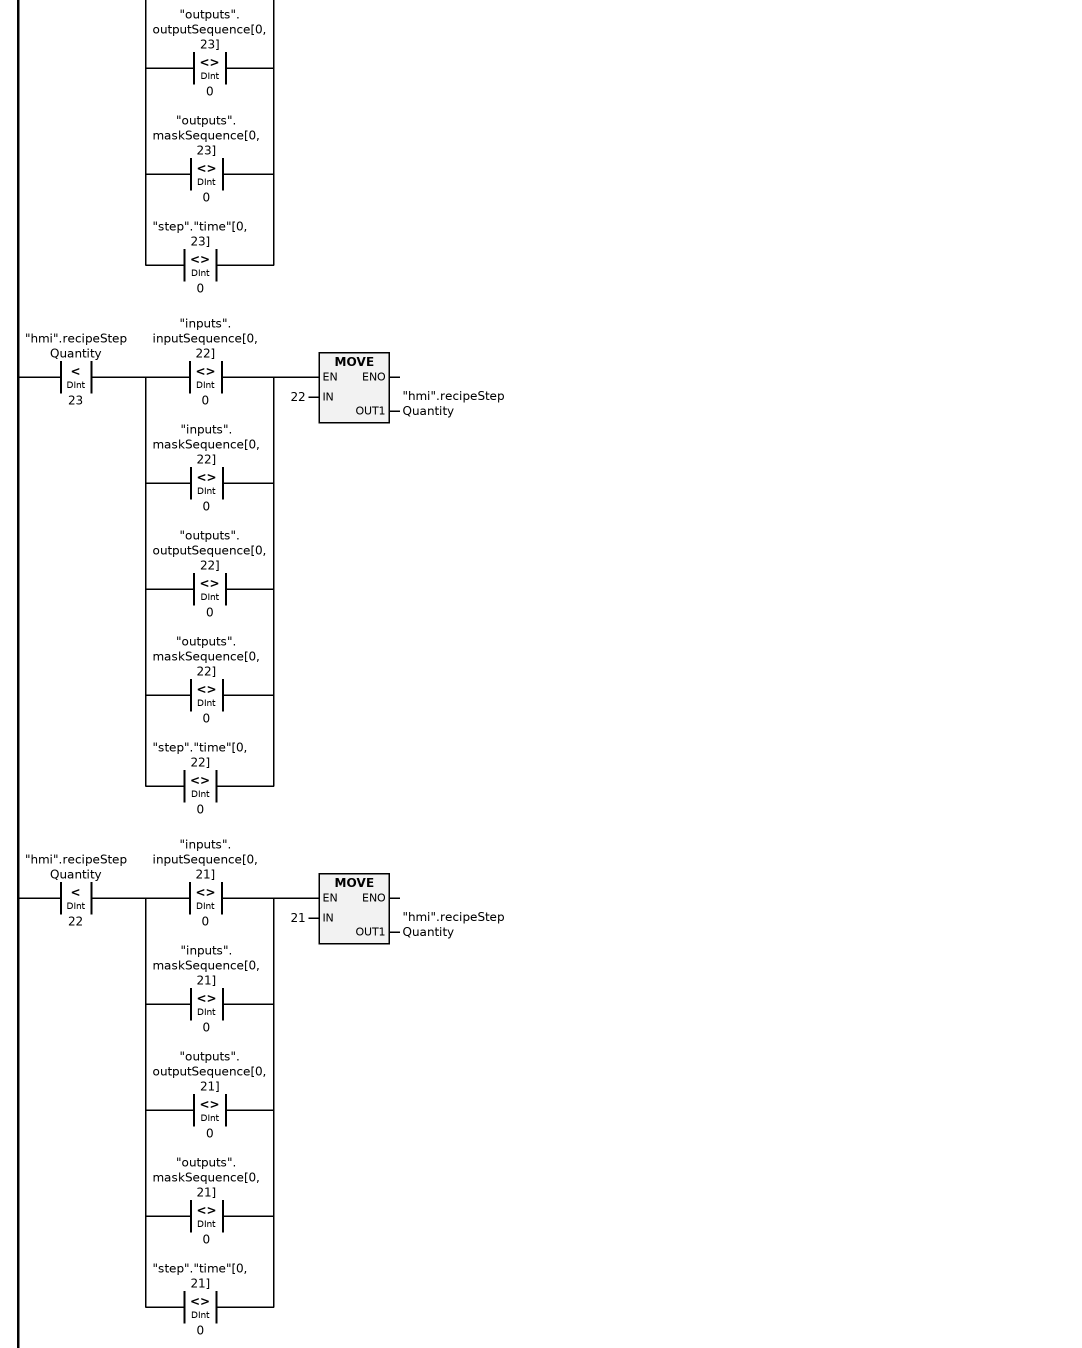
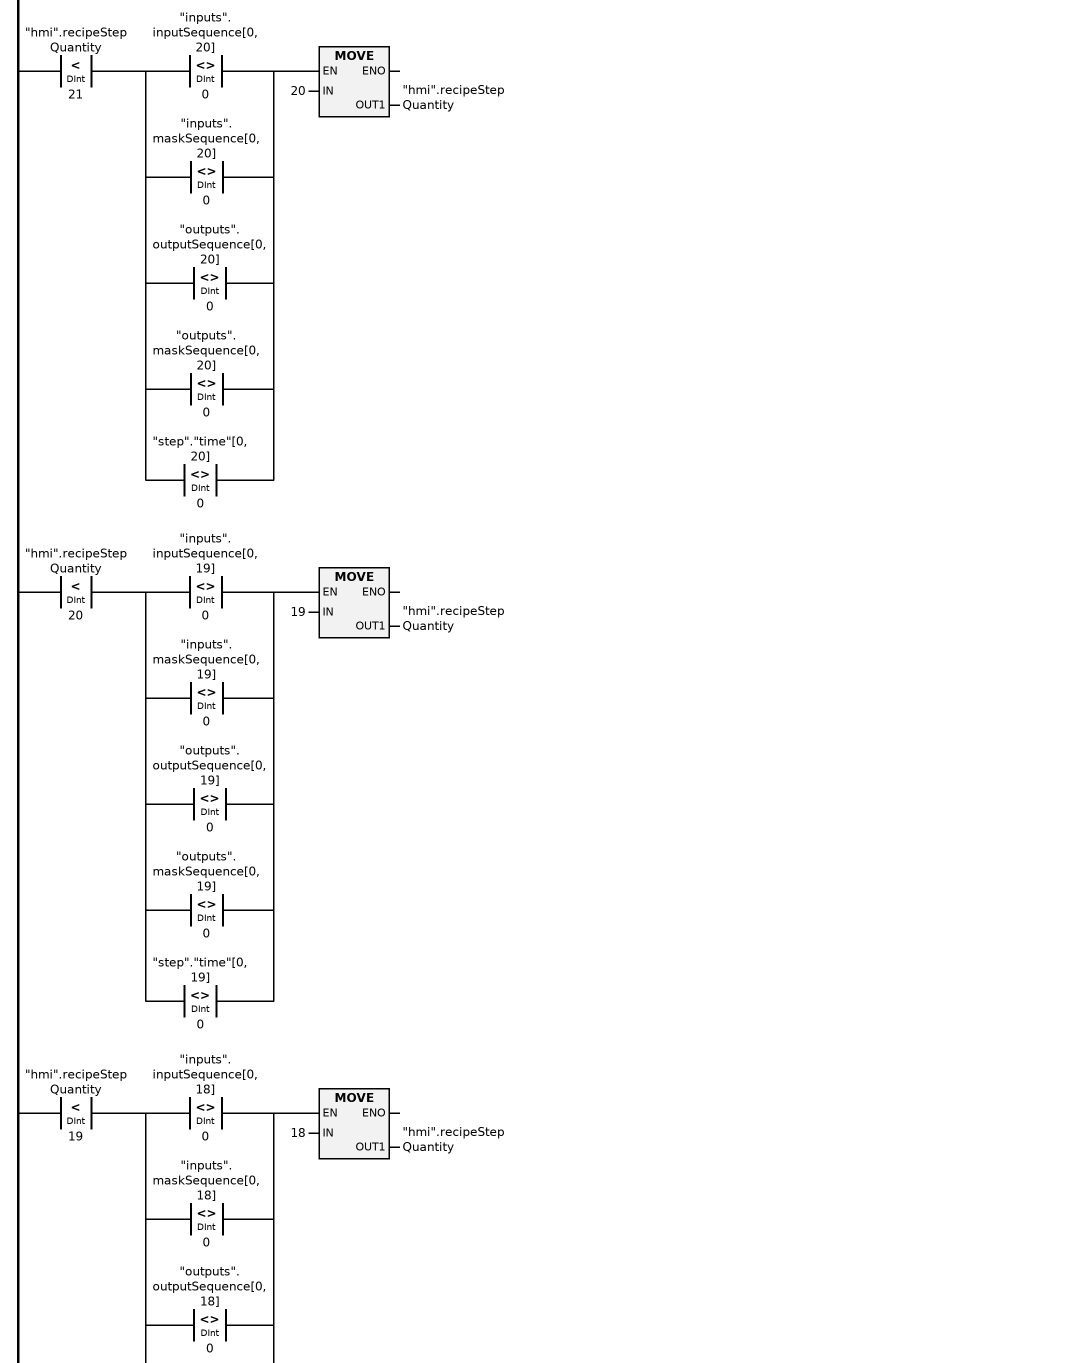
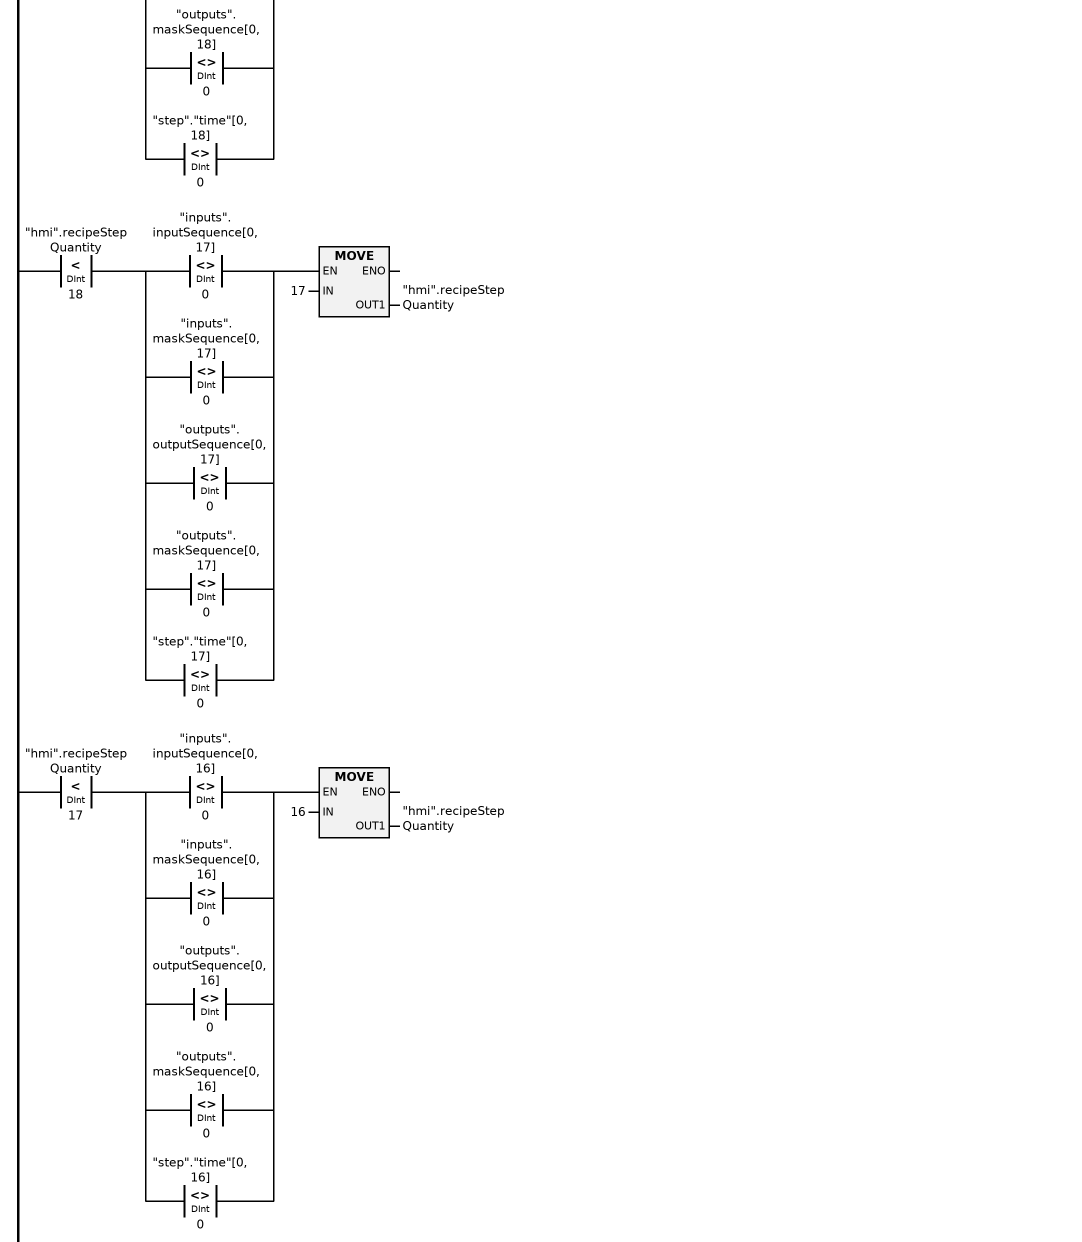
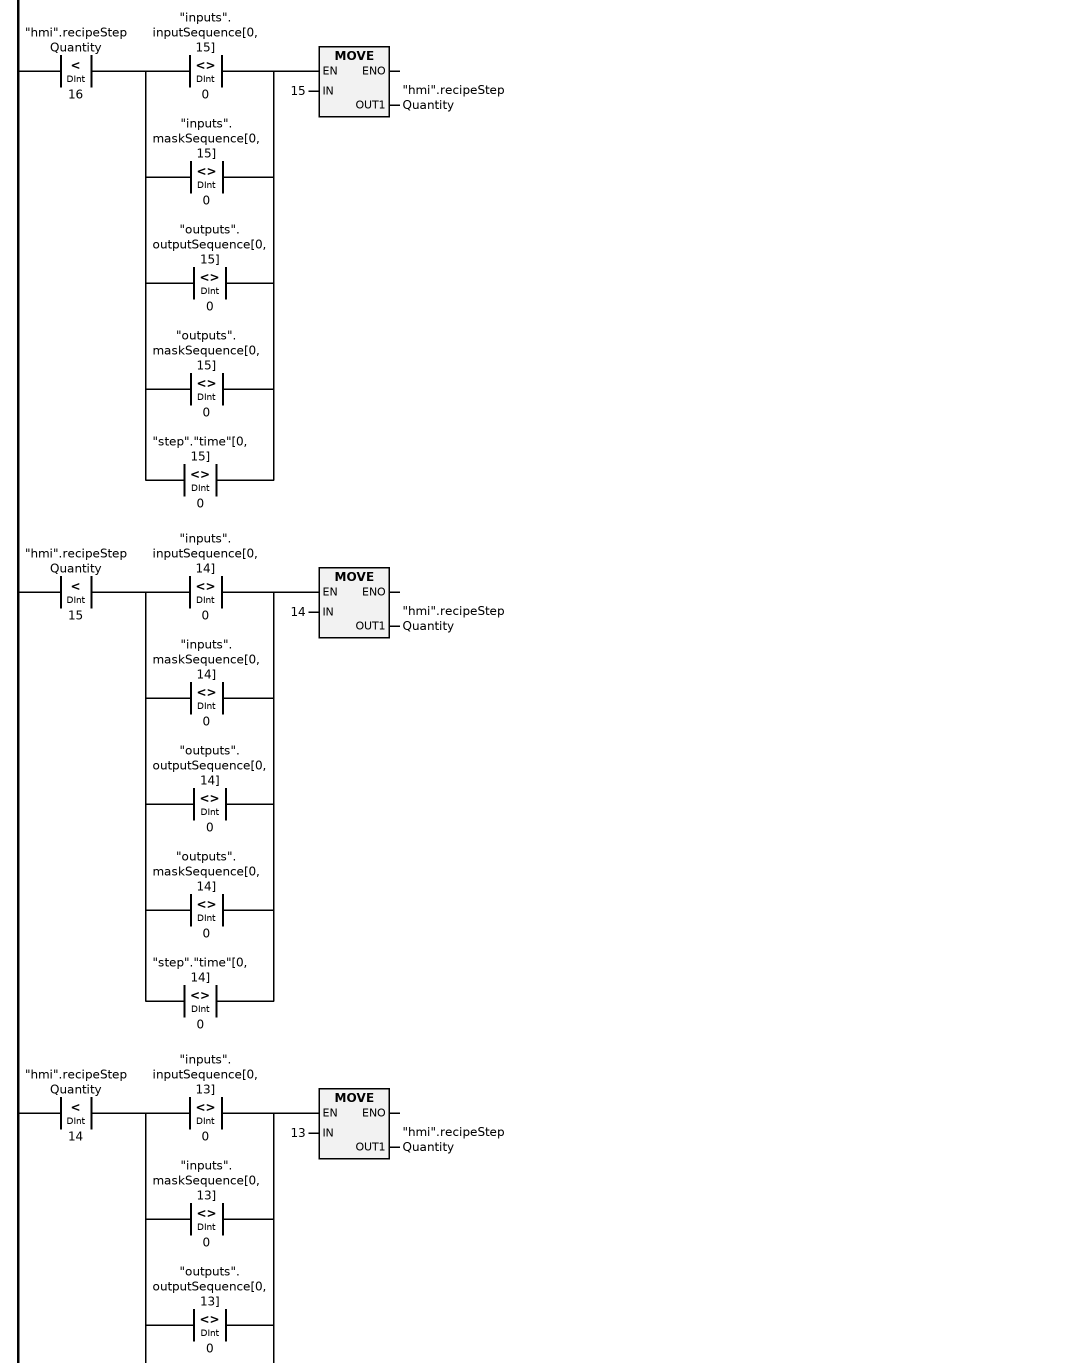
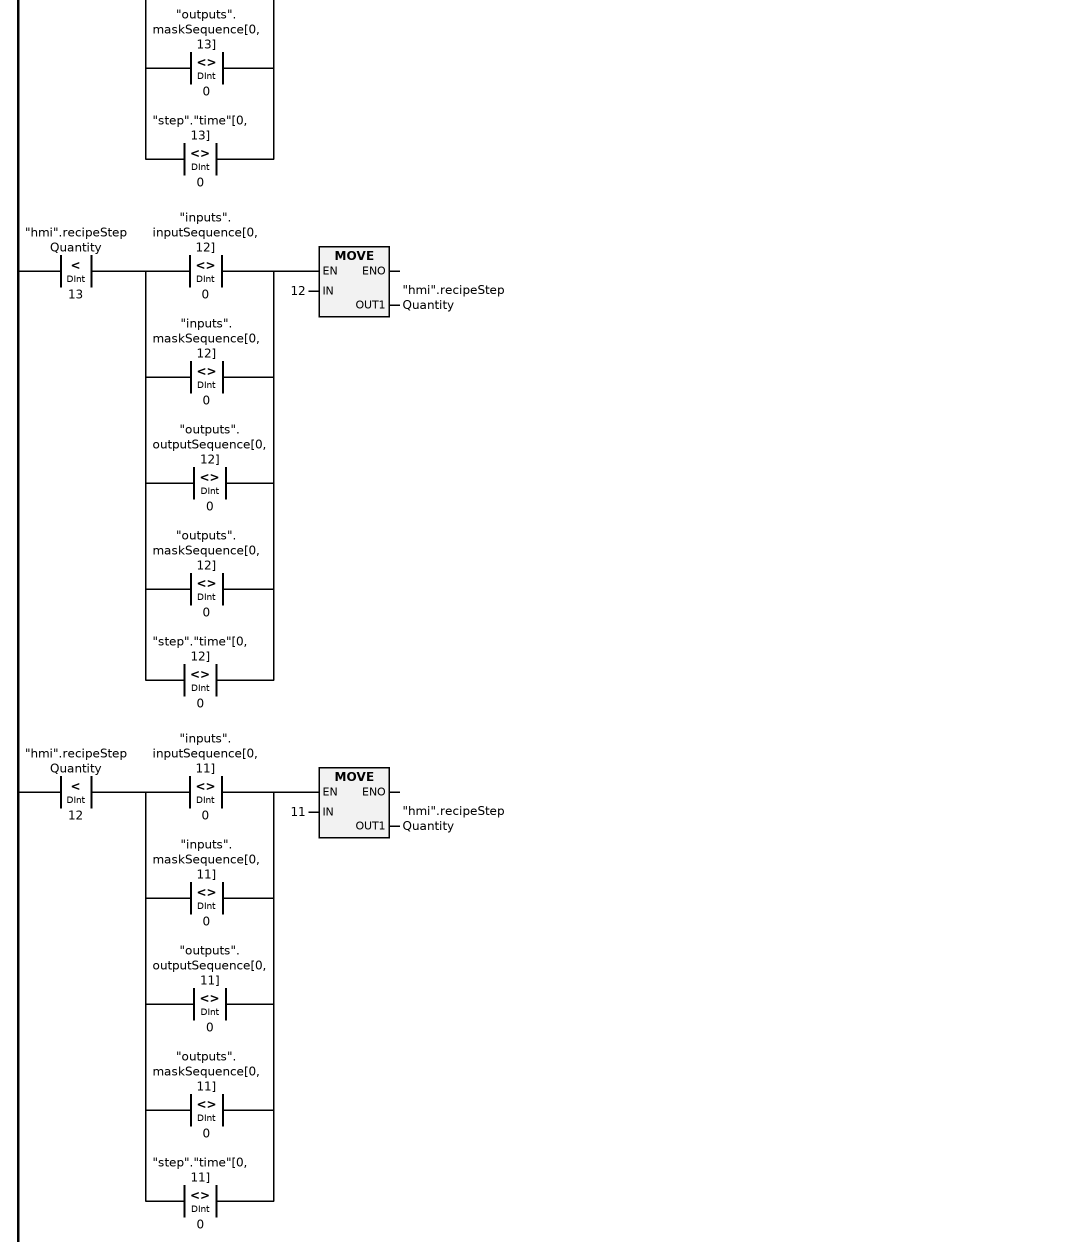
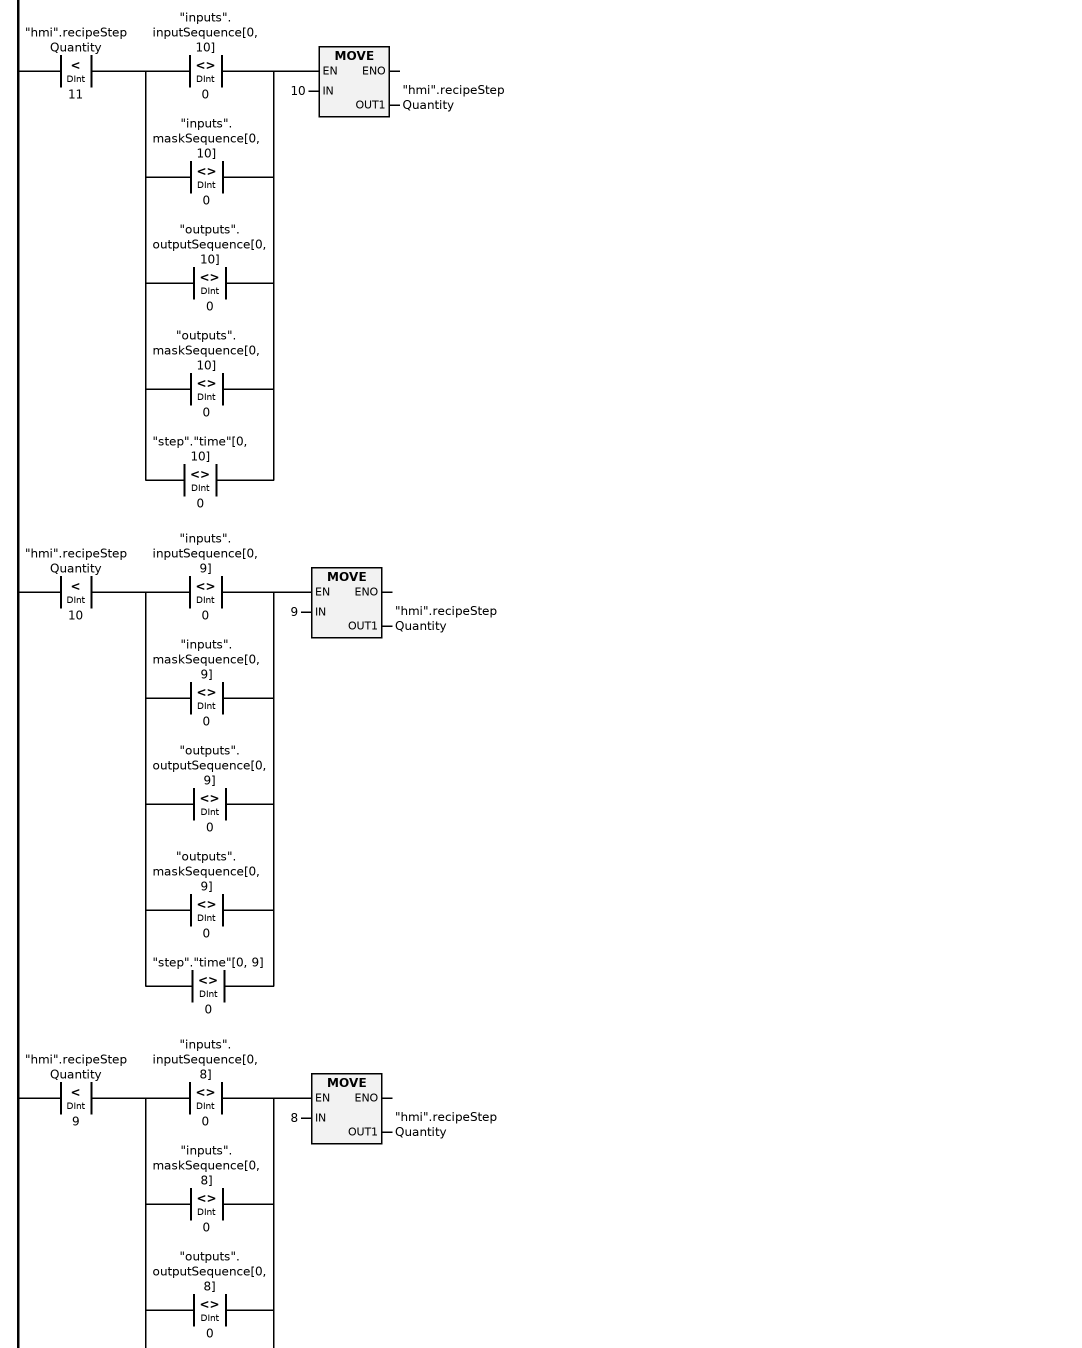
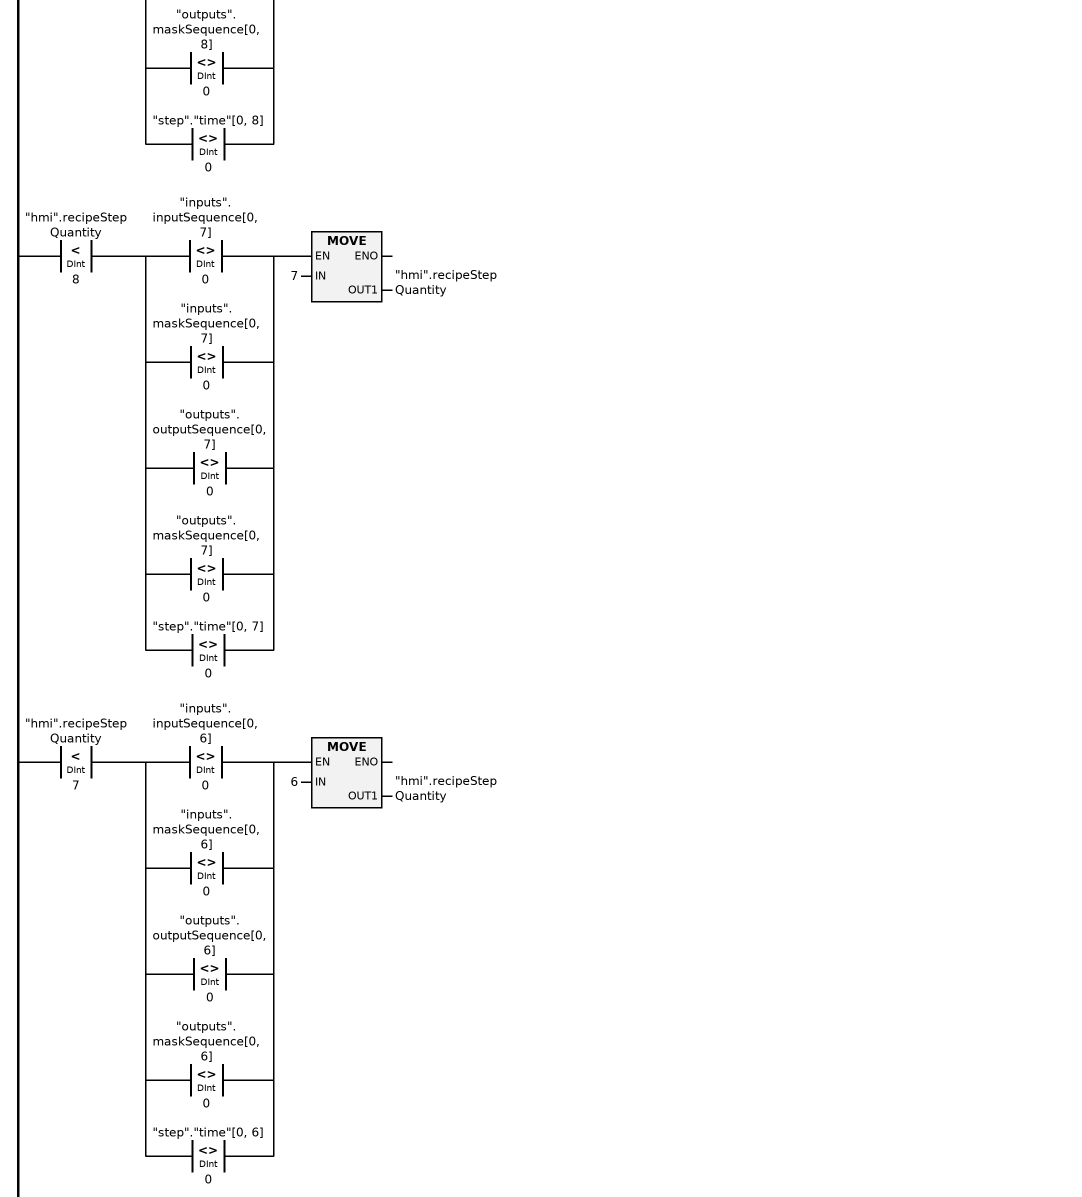
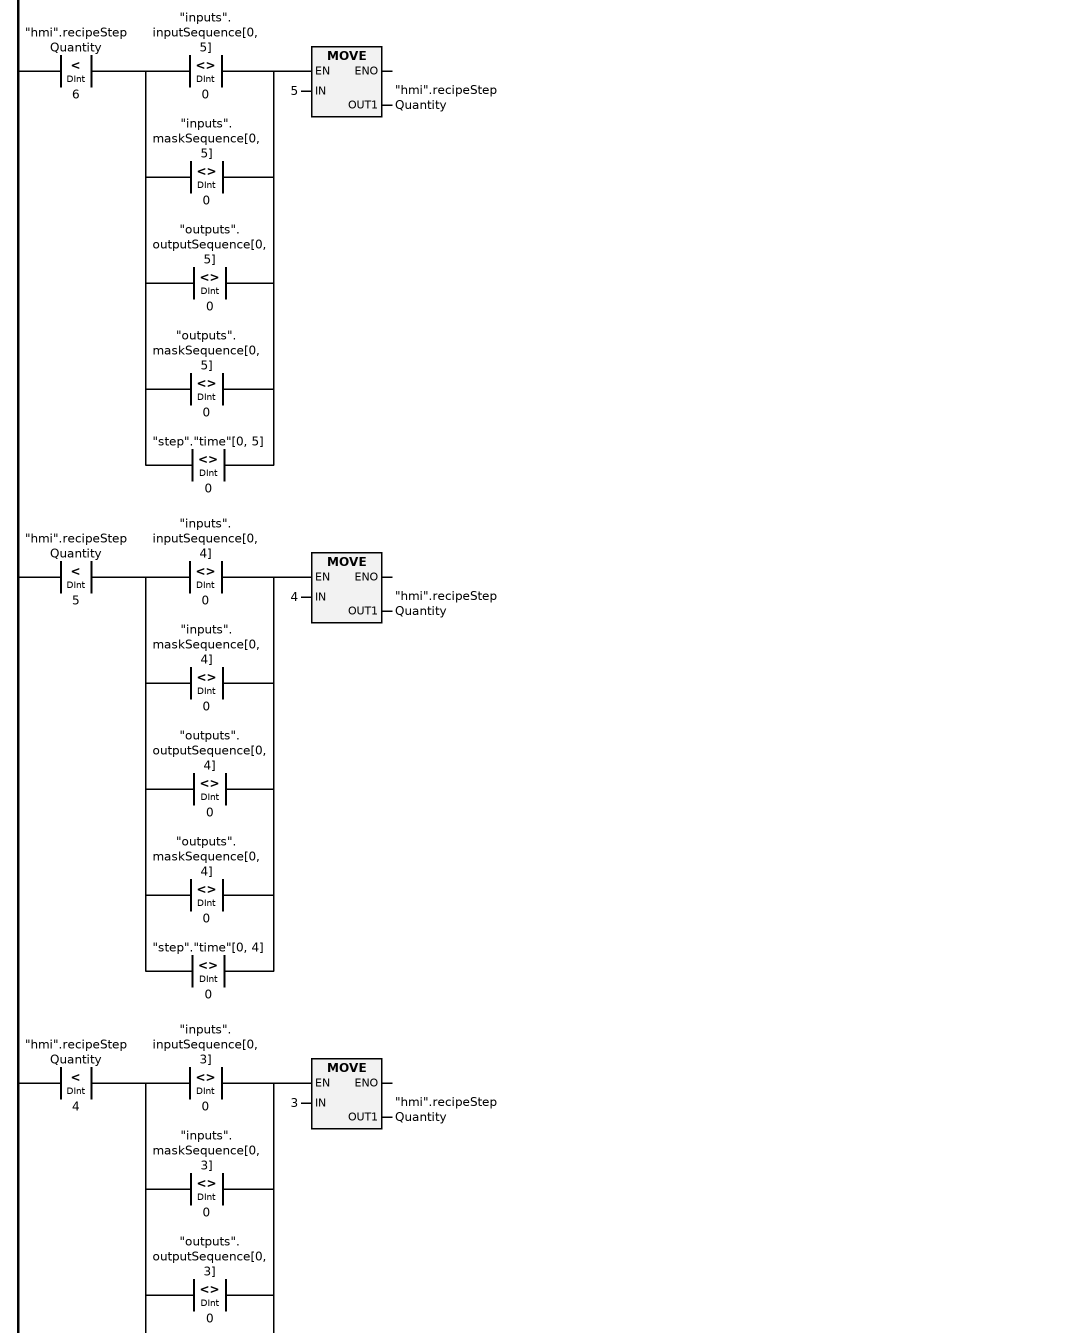
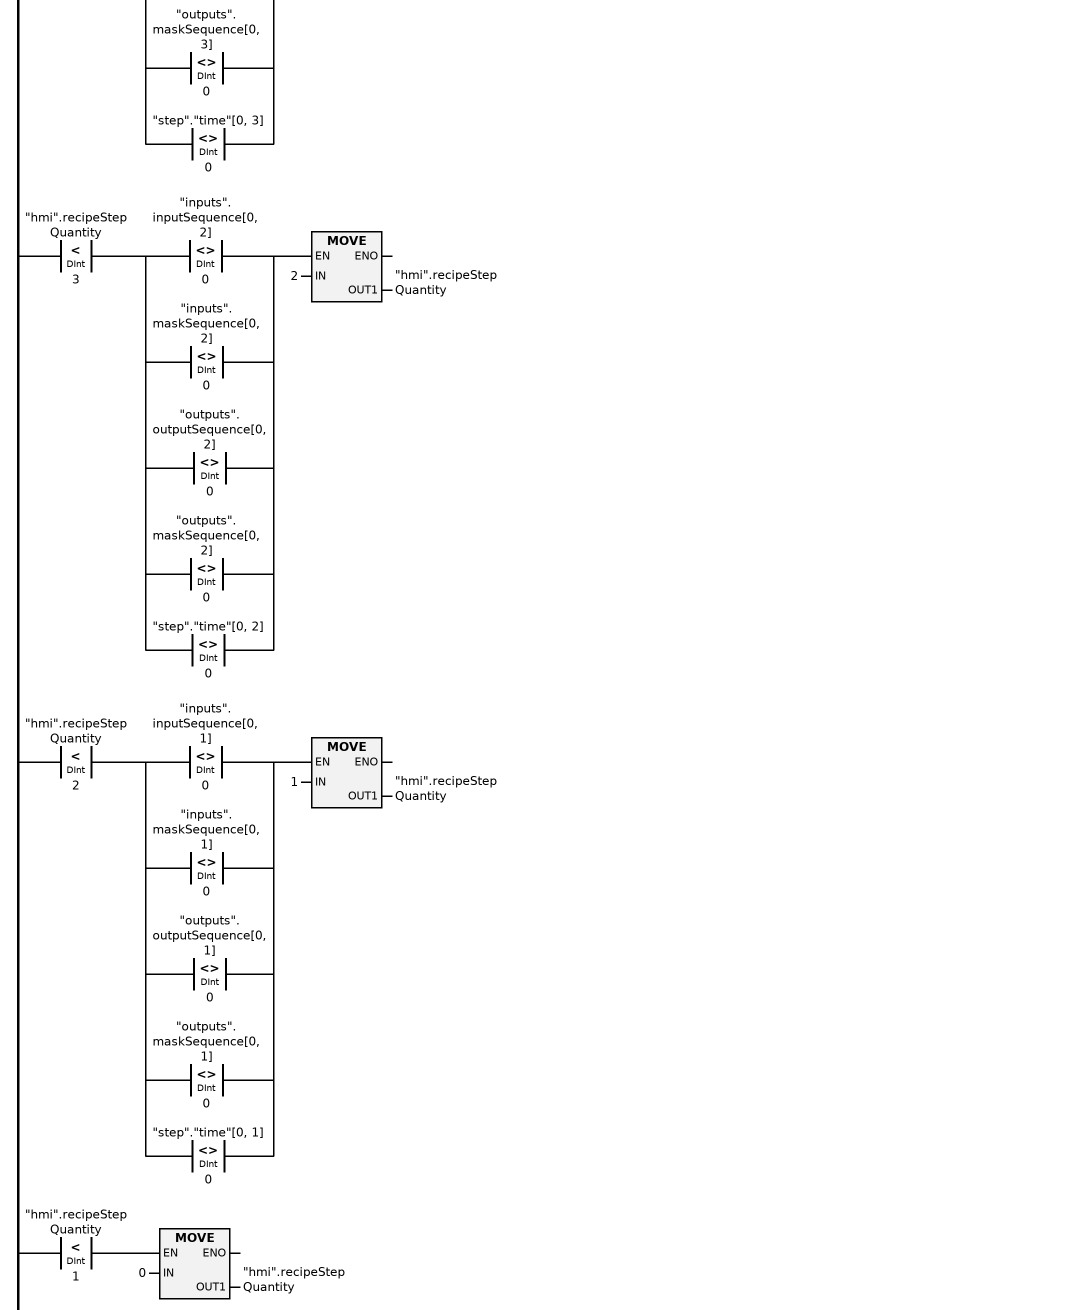
